KUKA KRL program: MyProgram_275().src

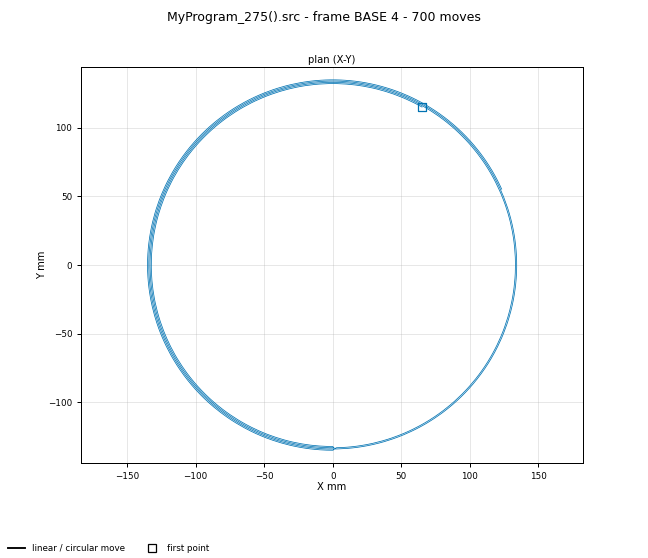
[picture p0: tool path of MyProgram_275().src in frame BASE 4, 700 of 700 moves have a stored position in this frame; points joined in program order, loops and branches not executed]
&ACCESS RVP
&REL 1
&PARAM TEMPLATE = C:\KRC\Roboter\Template\vorgabe
&PARAM EDITMASK = *
DEF MyProgram_275()
; ---- Setting reference (Base) ----
$BASE = BASE_DATA[4]

; --------------------------
; ---- Setting tool (TCP) ----
$TOOL = TOOL_DATA[3]
; --------------------------

$VEL.CP = VEL_APROX_PRINT
Startdeposition()
$VEL.CP = VEL_PRINT
LIN {X 65.127,Y 115.2291,Z 172,A 61.2414,B 9.2766,C 0.0638,E1 9.3556,E2 389.9841} C_DIS
LIN {X 62.4024,Y 116.727,Z 172,A 62.7582,B 9.2766,C 0.0584,E1 9.3518,E2 388.4469} C_DIS
LIN {X 59.3854,Y 118.2901,Z 172,A 64.0726,B 9.2766,C 0.0598,E1 9.3486,E2 387.151} C_DIS
LIN {X 56.4655,Y 119.7109,Z 172,A 65.4603,B 9.2766,C 0.0584,E1 9.3451,E2 385.7655} C_DIS
LIN {X 53.635,Y 121.0046,Z 172,A 66.8024,B 9.2766,C 0.0569,E1 9.3417,E2 384.424} C_DIS
LIN {X 50.5321,Y 122.3332,Z 172,A 68.2548,B 9.2766,C 0.0555,E1 9.3379,E2 382.9727} C_DIS
LIN {X 47.5119,Y 123.5374,Z 172,A 69.6526,B 9.2766,C 0.0543,E1 9.3343,E2 381.5762} C_DIS
LIN {X 44.4709,Y 124.6644,Z 172,A 71.05,B 9.2766,C 0.053,E1 9.3306,E2 380.1797} C_DIS
LIN {X 40.7766,Y 125.9215,Z 172,A 72.6186,B 9.2766,C 0.054,E1 9.3265,E2 378.6256} C_DIS
LIN {X 38.4338,Y 126.6555,Z 172,A 73.8215,B 9.2766,C 0.0503,E1 9.3232,E2 377.4063} C_DIS
LIN {X 35.3289,Y 127.5565,Z 172,A 75.1773,B 9.2766,C 0.0501,E1 9.3196,E2 376.056} C_DIS
LIN {X 32.2031,Y 128.3814,Z 172,A 76.5869,B 9.2767,C 0.0489,E1 9.3158,E2 374.6454} C_DIS
LIN {X 28.8757,Y 129.1715,Z 172,A 78.0434,B 9.2767,C 0.0484,E1 9.3118,E2 373.1922} C_DIS
LIN {X 25.6888,Y 129.8434,Z 172,A 79.4431,B 9.2767,C 0.0479,E1 9.308,E2 371.794} C_DIS
LIN {X 22.4953,Y 130.4347,Z 172,A 80.8231,B 9.2767,C 0.0477,E1 9.3042,E2 370.4175} C_DIS
LIN {X 19.425,Y 130.9271,Z 172,A 82.2366,B 9.2767,C 0.0458,E1 9.3003,E2 368.9965} C_DIS
LIN {X 16.2022,Y 131.364,Z 172,A 83.6161,B 9.2767,C 0.0458,E1 9.2965,E2 367.6208} C_DIS
LIN {X 12.5116,Y 131.7658,Z 172,A 85.1484,B 9.2767,C 0.0469,E1 9.2923,E2 366.0978} C_DIS
LIN {X 9.7365,Y 131.9999,Z 172,A 86.4152,B 9.2767,C 0.0455,E1 9.2887,E2 364.8243} C_DIS
LIN {X 6.4978,Y 132.199,Z 172,A 87.8269,B 9.2767,C 0.0451,E1 9.2848,E2 363.4123} C_DIS
LIN {X 3.2539,Y 132.3192,Z 172,A 89.2132,B 9.2767,C 0.0454,E1 9.2809,E2 362.0288} C_DIS
LIN {X 0.0153,Y 132.3605,Z 172,A 90.6902,B 9.2767,C 0.044,E1 9.2768,E2 360.5436} C_DIS
LIN {X -3.2492,Y 132.3193,Z 172,A 92.083,B 9.2767,C 0.0445,E1 9.2729,E2 359.1539} C_DIS
LIN {X -6.6259,Y 132.1926,Z 172,A 93.5018,B 9.2767,C 0.0456,E1 9.269,E2 357.7409} C_DIS
LIN {X -9.7303,Y 132.0004,Z 172,A 94.8665,B 9.2767,C 0.0456,E1 9.2651,E2 356.3748} C_DIS
LIN {X -13.1026,Y 131.7091,Z 172,A 96.308,B 9.2767,C 0.0464,E1 9.2612,E2 354.937} C_DIS
LIN {X -16.3389,Y 131.3477,Z 172,A 97.7167,B 9.2767,C 0.0469,E1 9.2572,E2 353.5291} C_DIS
LIN {X -19.5515,Y 130.9082,Z 172,A 99.1007,B 9.2767,C 0.0479,E1 9.2534,E2 352.1483} C_DIS
LIN {X -22.7528,Y 130.3893,Z 172,A 100.511,B 9.2767,C 0.0485,E1 9.2495,E2 350.7381} C_DIS
LIN {X -26.0765,Y 129.7645,Z 172,A 101.9358,B 9.2767,C 0.0501,E1 9.2457,E2 349.3187} C_DIS
LIN {X -29.4885,Y 129.0315,Z 172,A 103.4456,B 9.2767,C 0.0511,E1 9.2415,E2 347.81} C_DIS
LIN {X -32.29,Y 128.3594,Z 172,A 104.7854,B 9.2767,C 0.0503,E1 9.2379,E2 346.4602} C_DIS
LIN {X -35.9173,Y 127.392,Z 172,A 106.3281,B 9.2767,C 0.0531,E1 9.2338,E2 344.9283} C_DIS
LIN {X -38.4302,Y 126.6566,Z 172,A 107.5882,B 9.2767,C 0.0517,E1 9.2303,E2 343.654} C_DIS
LIN {X -41.6366,Y 125.6388,Z 172,A 108.9857,B 9.2767,C 0.0541,E1 9.2266,E2 342.2646} C_DIS
LIN {X -44.5824,Y 124.6241,Z 172,A 110.3733,B 9.2767,C 0.0548,E1 9.223,E2 340.8734} C_DIS
LIN {X -47.6183,Y 123.4961,Z 172,A 111.7823,B 9.2767,C 0.0561,E1 9.2193,E2 339.4646} C_DIS
LIN {X -50.7473,Y 122.2434,Z 172,A 113.2597,B 9.2767,C 0.0574,E1 9.2155,E2 337.9861} C_DIS
LIN {X -53.7595,Y 120.9489,Z 172,A 114.6384,B 9.2767,C 0.0598,E1 9.212,E2 336.6133} C_DIS
LIN {X -56.5897,Y 119.6516,Z 172,A 116.0384,B 9.2767,C 0.0606,E1 9.2084,E2 335.2083} C_DIS
LIN {X -59.5181,Y 118.2226,Z 172,A 117.496,B 9.2767,C 0.0616,E1 9.2048,E2 333.7464} C_DIS
LIN {X -62.5135,Y 116.6673,Z 172,A 118.9788,B 9.2767,C 0.0633,E1 9.2011,E2 332.2623} C_DIS
LIN {X -65.2363,Y 115.1675,Z 172,A 120.2908,B 9.2766,C 0.0658,E1 9.1979,E2 330.9554} C_DIS
LIN {X -68.1488,Y 113.4684,Z 172,A 121.7627,B 9.2766,C 0.0678,E1 9.1944,E2 329.4833} C_DIS
LIN {X -70.9084,Y 111.7643,Z 172,A 123.1624,B 9.2766,C 0.0701,E1 9.1911,E2 328.0853} C_DIS
LIN {X -74.0157,Y 109.731,Z 172,A 124.7159,B 9.2766,C 0.0736,E1 9.1875,E2 326.5396} C_DIS
LIN {X -76.2793,Y 108.1694,Z 172,A 125.9901,B 9.2766,C 0.0742,E1 9.1845,E2 325.2566} C_DIS
LIN {X -78.717,Y 106.4094,Z 172,A 127.4521,B 9.2766,C 0.0737,E1 9.1812,E2 323.7769} C_DIS
LIN {X -82.0673,Y 103.8473,Z 172,A 129.3252,B 9.2766,C 0.0762,E1 9.1771,E2 321.9} C_DIS
LIN {X -85.2696,Y 101.234,Z 172,A 131.1208,B 9.2765,C 0.0795,E1 9.1732,E2 320.1053} C_DIS
LIN {X -88.3376,Y 98.5679,Z 172,A 132.89,B 9.2765,C 0.0828,E1 9.1695,E2 318.3366} C_DIS
LIN {X -91.8024,Y 95.35,Z 172,A 134.8455,B 9.2765,C 0.0885,E1 9.1656,E2 316.3939} C_DIS
LIN {X -94.7344,Y 92.4374,Z 172,A 136.7676,B 9.2764,C 0.0899,E1 9.1618,E2 314.4579} C_DIS
LIN {X -97.5284,Y 89.484,Z 172,A 138.5544,B 9.2764,C 0.0933,E1 9.1584,E2 312.6697} C_DIS
LIN {X -100.2218,Y 86.4567,Z 172,A 140.3227,B 9.2764,C 0.0969,E1 9.1551,E2 310.9015} C_DIS
LIN {X -102.8625,Y 83.2979,Z 172,A 142.1311,B 9.2763,C 0.1005,E1 9.1519,E2 309.0918} C_DIS
LIN {X -105.4209,Y 80.0359,Z 172,A 143.7918,B 9.2763,C 0.107,E1 9.1491,E2 307.4488} C_DIS
LIN {X -107.2971,Y 77.5019,Z 172,A 145.1917,B 9.2762,C 0.1096,E1 9.1468,E2 306.0461} C_DIS
LIN {X -109.1538,Y 74.864,Z 172,A 146.6295,B 9.2762,C 0.1123,E1 9.1445,E2 304.6049} C_DIS
LIN {X -110.9486,Y 72.1775,Z 172,A 148.1,B 9.2762,C 0.1145,E1 9.1422,E2 303.1273} C_DIS
LIN {X -112.6772,Y 69.4484,Z 172,A 149.4685,B 9.2761,C 0.1185,E1 9.1402,E2 301.7638} C_DIS
LIN {X -114.4012,Y 66.5704,Z 172,A 150.9053,B 9.2761,C 0.1224,E1 9.1382,E2 300.3303} C_DIS
LIN {X -115.9291,Y 63.8724,Z 172,A 152.2877,B 9.276,C 0.1252,E1 9.1363,E2 298.9445} C_DIS
LIN {X -117.5491,Y 60.8396,Z 172,A 153.7952,B 9.276,C 0.1288,E1 9.1343,E2 297.4364} C_DIS
LIN {X -119.004,Y 57.941,Z 172,A 155.2177,B 9.2759,C 0.1321,E1 9.1326,E2 296.0131} C_DIS
LIN {X -120.3328,Y 55.1259,Z 172,A 156.5823,B 9.2759,C 0.1354,E1 9.131,E2 294.6479} C_DIS
LIN {X -121.6532,Y 52.1471,Z 172,A 158.0257,B 9.2759,C 0.1387,E1 9.1294,E2 293.2021} C_DIS
LIN {X -122.9461,Y 49.0219,Z 172,A 159.5002,B 9.2757,C 0.1425,E1 9.1278,E2 291.7279} C_DIS
LIN {X -124.1154,Y 45.981,Z 172,A 160.93,B 9.2757,C 0.146,E1 9.1264,E2 290.2972} C_DIS
LIN {X -125.2045,Y 42.9266,Z 172,A 162.3419,B 9.2757,C 0.1498,E1 9.1251,E2 288.8858} C_DIS
LIN {X -126.34,Y 39.4647,Z 172,A 163.9378,B 9.2756,C 0.1539,E1 9.1237,E2 287.2894} C_DIS
LIN {X -127.1202,Y 36.868,Z 172,A 165.147,B 9.2756,C 0.1566,E1 9.1228,E2 286.0771} C_DIS
LIN {X -127.9856,Y 33.7419,Z 172,A 166.5722,B 9.2755,C 0.1602,E1 9.1217,E2 284.6509} C_DIS
LIN {X -128.8049,Y 30.4681,Z 172,A 168.0566,B 9.2754,C 0.164,E1 9.1208,E2 283.1651} C_DIS
LIN {X -129.5239,Y 27.2532,Z 172,A 169.5788,B 9.2754,C 0.1665,E1 9.1199,E2 281.633} C_DIS
LIN {X -130.1092,Y 24.303,Z 172,A 170.8243,B 9.2753,C 0.1711,E1 9.1192,E2 280.3955} C_DIS
LIN {X -130.6809,Y 21.0199,Z 172,A 172.3104,B 9.2753,C 0.1746,E1 9.1185,E2 278.9057} C_DIS
LIN {X -131.1563,Y 17.8087,Z 172,A 173.7369,B 9.2751,C 0.1783,E1 9.118,E2 277.478} C_DIS
LIN {X -131.5527,Y 14.5881,Z 172,A 175.163,B 9.2751,C 0.182,E1 9.1175,E2 276.0508} C_DIS
LIN {X -131.8826,Y 11.214,Z 172,A 176.6177,B 9.275,C 0.1865,E1 9.1171,E2 274.599} C_DIS
LIN {X -132.1096,Y 8.1125,Z 172,A 178.0102,B 9.275,C 0.1896,E1 9.1169,E2 273.2023} C_DIS
LIN {X -132.2745,Y 4.7345,Z 172,A 179.4735,B 9.2748,C 0.1939,E1 9.1167,E2 271.7405} C_DIS
LIN {X -132.3534,Y 1.3457,Z 172,A -179.134,B 9.2748,C 0.1994,E1 9.1167,E2 270.3584} C_DIS
LIN {X -132.3475,Y -1.7648,Z 172,A -177.662,B 9.2747,C 0.2013,E1 9.1167,E2 268.8726} C_DIS
LIN {X -132.2638,Y -5.0086,Z 172,A -176.2074,B 9.2746,C 0.2045,E1 9.1167,E2 267.4133} C_DIS
LIN {X -132.0874,Y -8.4737,Z 172,A -174.7375,B 9.2745,C 0.2094,E1 9.117,E2 265.9486} C_DIS
LIN {X -131.8595,Y -11.4869,Z 172,A -173.3647,B 9.2745,C 0.2121,E1 9.1173,E2 264.5693} C_DIS
LIN {X -131.4649,Y -15.3568,Z 172,A -171.8356,B 9.2743,C 0.2195,E1 9.1178,E2 263.0602} C_DIS
LIN {X -131.1377,Y -17.9505,Z 172,A -170.4833,B 9.2743,C 0.2192,E1 9.1183,E2 261.6826} C_DIS
LIN {X -130.679,Y -21.0311,Z 172,A -169.0538,B 9.2743,C 0.2217,E1 9.1189,E2 260.2445} C_DIS
LIN {X -130.1175,Y -24.2591,Z 172,A -167.6784,B 9.2741,C 0.2264,E1 9.1196,E2 258.8755} C_DIS
LIN {X -129.4878,Y -27.4207,Z 172,A -166.2107,B 9.2741,C 0.2292,E1 9.1204,E2 257.4002} C_DIS
LIN {X -128.7496,Y -30.6976,Z 172,A -164.7876,B 9.2739,C 0.2338,E1 9.1213,E2 255.982} C_DIS
LIN {X -127.9636,Y -33.8244,Z 172,A -163.372,B 9.2739,C 0.2373,E1 9.1223,E2 254.5651} C_DIS
LIN {X -127.1019,Y -36.9304,Z 172,A -161.8377,B 9.2738,C 0.2389,E1 9.1235,E2 253.0151} C_DIS
LIN {X -125.7599,Y -41.2728,Z 172,A -159.8805,B 9.2736,C 0.2445,E1 9.1252,E2 251.0607} C_DIS
LIN {X -124.439,Y -45.0958,Z 172,A -158.2958,B 9.2734,C 0.252,E1 9.1266,E2 249.4973} C_DIS
LIN {X -123.3976,Y -47.8715,Z 172,A -156.8678,B 9.2734,C 0.253,E1 9.128,E2 248.0528} C_DIS
LIN {X -122.2317,Y -50.7753,Z 172,A -155.5005,B 9.2734,C 0.2564,E1 9.1295,E2 246.6849} C_DIS
LIN {X -120.9497,Y -53.7578,Z 172,A -154.0011,B 9.2733,C 0.2585,E1 9.1312,E2 245.1751} C_DIS
LIN {X -119.6466,Y -56.6002,Z 172,A -152.7067,B 9.2731,C 0.263,E1 9.1327,E2 243.8888} C_DIS
LIN {X -118.2264,Y -59.5107,Z 172,A -151.243,B 9.2731,C 0.2656,E1 9.1345,E2 242.4185} C_DIS
LIN {X -116.6748,Y -62.4995,Z 172,A -149.8397,B 9.2729,C 0.2702,E1 9.1363,E2 241.0228} C_DIS
LIN {X -115.1644,Y -65.2418,Z 172,A -148.4248,B 9.2729,C 0.2726,E1 9.1383,E2 239.6015} C_DIS
LIN {X -113.4581,Y -68.1657,Z 172,A -146.9417,B 9.2728,C 0.2759,E1 9.1404,E2 238.1171} C_DIS
LIN {X -111.7542,Y -70.9245,Z 172,A -145.3675,B 9.2728,C 0.2764,E1 9.1428,E2 236.523} C_DIS
LIN {X -109.9736,Y -73.6546,Z 172,A -144.085,B 9.2726,C 0.2819,E1 9.1447,E2 235.2568} C_DIS
LIN {X -107.9412,Y -76.6029,Z 172,A -142.5621,B 9.2725,C 0.2859,E1 9.1471,E2 233.738} C_DIS
LIN {X -106.316,Y -78.8425,Z 172,A -141.167,B 9.2725,C 0.2853,E1 9.1495,E2 232.3195} C_DIS
LIN {X -103.8545,Y -82.0582,Z 172,A -139.3643,B 9.2724,C 0.2884,E1 9.1526,E2 230.5116} C_DIS
LIN {X -101.2348,Y -85.2687,Z 172,A -137.5611,B 9.2723,C 0.2921,E1 9.1558,E2 228.708} C_DIS
LIN {X -98.5714,Y -88.3337,Z 172,A -135.9358,B 9.2721,C 0.2981,E1 9.1588,E2 227.0996} C_DIS
LIN {X -95.8719,Y -91.2568,Z 172,A -134.0515,B 9.2721,C 0.2988,E1 9.1624,E2 225.1962} C_DIS
LIN {X -92.9642,Y -94.2177,Z 172,A -132.2243,B 9.272,C 0.3018,E1 9.166,E2 223.3658} C_DIS
LIN {X -90.0913,Y -96.9677,Z 172,A -130.4908,B 9.2719,C 0.3049,E1 9.1696,E2 221.6314} C_DIS
LIN {X -87.0184,Y -99.7345,Z 172,A -128.7007,B 9.2718,C 0.3082,E1 9.1733,E2 219.8418} C_DIS
LIN {X -83.9207,Y -102.3549,Z 172,A -126.9148,B 9.2717,C 0.3108,E1 9.1772,E2 218.0527} C_DIS
LIN {X -80.3433,Y -105.1862,Z 172,A -125.0181,B 9.2715,C 0.3155,E1 9.1813,E2 216.166} C_DIS
LIN {X -77.5467,Y -107.2646,Z 172,A -123.5366,B 9.2715,C 0.3184,E1 9.1847,E2 214.6881} C_DIS
LIN {X -74.901,Y -109.1284,Z 172,A -122.1001,B 9.2714,C 0.32,E1 9.188,E2 213.2474} C_DIS
LIN {X -71.9097,Y -111.1224,Z 172,A -120.6166,B 9.2712,C 0.3236,E1 9.1914,E2 211.773} C_DIS
LIN {X -69.4334,Y -112.6864,Z 172,A -119.2487,B 9.2712,C 0.3236,E1 9.1947,E2 210.393} C_DIS
LIN {X -66.5381,Y -114.4199,Z 172,A -117.8103,B 9.2712,C 0.3261,E1 9.1981,E2 208.9574} C_DIS
LIN {X -63.0793,Y -116.3627,Z 172,A -115.9086,B 9.2712,C 0.3249,E1 9.2028,E2 207.0333} C_DIS
LIN {X -59.1058,Y -118.4294,Z 172,A -114.2002,B 9.271,C 0.3315,E1 9.207,E2 205.3531} C_DIS
LIN {X -56.4686,Y -119.7095,Z 172,A -112.8473,B 9.271,C 0.3315,E1 9.2104,E2 203.9899} C_DIS
LIN {X -53.6395,Y -121.0027,Z 172,A -111.4883,B 9.271,C 0.3326,E1 9.2139,E2 202.6293} C_DIS
LIN {X -50.5291,Y -122.3345,Z 172,A -110.0165,B 9.2709,C 0.334,E1 9.2177,E2 201.1565} C_DIS
LIN {X -47.5164,Y -123.5357,Z 172,A -108.603,B 9.2709,C 0.3351,E1 9.2214,E2 199.7417} C_DIS
LIN {X -43.7679,Y -124.9129,Z 172,A -107.016,B 9.2707,C 0.3393,E1 9.2255,E2 198.1718} C_DIS
LIN {X -41.5296,Y -125.6744,Z 172,A -105.8276,B 9.2707,C 0.337,E1 9.2287,E2 196.9631} C_DIS
LIN {X -38.447,Y -126.6515,Z 172,A -104.4389,B 9.2707,C 0.3383,E1 9.2324,E2 195.5755} C_DIS
LIN {X -35.3408,Y -127.5532,Z 172,A -103.029,B 9.2707,C 0.339,E1 9.2362,E2 194.1642} C_DIS
LIN {X -32.1624,Y -128.3918,Z 172,A -101.5669,B 9.2707,C 0.3392,E1 9.2402,E2 192.6969} C_DIS
LIN {X -28.8672,Y -129.1734,Z 172,A -100.1405,B 9.2707,C 0.3407,E1 9.244,E2 191.2751} C_DIS
LIN {X -25.6893,Y -129.8433,Z 172,A -98.736,B 9.2707,C 0.3414,E1 9.2479,E2 189.8703} C_DIS
LIN {X -22.5021,Y -130.4336,Z 172,A -97.3492,B 9.2706,C 0.3422,E1 9.2517,E2 188.4852} C_DIS
LIN {X -19.4209,Y -130.9277,Z 172,A -95.9517,B 9.2706,C 0.3418,E1 9.2556,E2 187.0814} C_DIS
LIN {X -16.1963,Y -131.3647,Z 172,A -94.5436,B 9.2706,C 0.3421,E1 9.2595,E2 185.6729} C_DIS
LIN {X -12.9725,Y -131.7216,Z 172,A -93.1122,B 9.2706,C 0.3418,E1 9.2635,E2 184.2377} C_DIS
LIN {X -9.7403,Y -131.9996,Z 172,A -91.7423,B 9.2706,C 0.3427,E1 9.2673,E2 182.8714} C_DIS
LIN {X -6.5025,Y -132.1988,Z 172,A -90.3296,B 9.2706,C 0.3426,E1 9.2712,E2 181.4571} C_DIS
LIN {X -3.2603,Y -132.319,Z 172,A -88.9419,B 9.2706,C 0.3428,E1 9.2751,E2 180.0709} C_DIS
LIN {X 0.0022,Y -132.3606,Z 172,A -87.4599,B 9.2706,C 0.3413,E1 9.2792,E2 178.5796} C_DIS
LIN {X 0.0022,Y -132.3606,Z 172,A -87.4599,B 9.2706,C 0.3413,E1 9.2792,E2 178.5796} C_DIS
Enddeposition()
LIN {X 0.9646,Y -133.2632,Z 172,A -87.4493,B 9.2704,C 0.3548,E1 9.2793,E2 178.6525} C_DIS
Startdeposition()
$VEL.CP = VEL_PRINT
LIN {X -2.4756,Y -133.245,Z 172,A -89.1713,B 9.2702,C 0.3597,E1 9.2744,E2 180.4051} C_DIS
LIN {X -6.4739,Y -133.1105,Z 172,A -90.8363,B 9.2702,C 0.3587,E1 9.2698,E2 182.0641} C_DIS
LIN {X -9.0906,Y -132.9586,Z 172,A -91.9518,B 9.2702,C 0.3584,E1 9.2667,E2 183.1787} C_DIS
LIN {X -11.5379,Y -132.7676,Z 172,A -93.049,B 9.2702,C 0.3591,E1 9.2636,E2 184.2814} C_DIS
LIN {X -14.6359,Y -132.462,Z 172,A -94.5024,B 9.2702,C 0.3611,E1 9.2595,E2 185.7494} C_DIS
LIN {X -18.1761,Y -132.0239,Z 172,A -95.9099,B 9.2702,C 0.3582,E1 9.2557,E2 187.142} C_DIS
LIN {X -21.515,Y -131.52,Z 172,A -97.4529,B 9.2702,C 0.3595,E1 9.2514,E2 188.6966} C_DIS
LIN {X -25.559,Y -130.7947,Z 172,A -99.3204,B 9.2702,C 0.3607,E1 9.2462,E2 190.577} C_DIS
LIN {X -29.5392,Y -129.9525,Z 172,A -100.9567,B 9.2702,C 0.3577,E1 9.2418,E2 192.2} C_DIS
LIN {X -33.0336,Y -129.1086,Z 172,A -102.5702,B 9.2702,C 0.3581,E1 9.2374,E2 193.8222} C_DIS
LIN {X -39.108,Y -127.4,Z 172,A -105.3268,B 9.2702,C 0.357,E1 9.23,E2 196.5845} C_DIS
LIN {X -42.5916,Y -126.279,Z 172,A -106.9251,B 9.2703,C 0.3563,E1 9.2257,E2 198.1862} C_DIS
LIN {X -47.3324,Y -124.5801,Z 172,A -108.9509,B 9.2705,C 0.3517,E1 9.2205,E2 200.1953} C_DIS
LIN {X -49.7048,Y -123.6511,Z 172,A -109.9688,B 9.2705,C 0.3492,E1 9.2179,E2 201.2037} C_DIS
LIN {X -52.1729,Y -122.6325,Z 172,A -111.2112,B 9.2705,C 0.3498,E1 9.2146,E2 202.4578} C_DIS
LIN {X -56.5524,Y -120.6749,Z 172,A -113.3293,B 9.2706,C 0.3486,E1 9.2092,E2 204.5828} C_DIS
LIN {X -61.9383,Y -117.999,Z 172,A -115.716,B 9.2709,C 0.3419,E1 9.2033,E2 206.9452} C_DIS
LIN {X -64.4835,Y -116.63,Z 172,A -117.2749,B 9.2707,C 0.346,E1 9.1994,E2 208.5427} C_DIS
LIN {X -68.5645,Y -114.2792,Z 172,A -119.1647,B 9.2709,C 0.3408,E1 9.1949,E2 210.4159} C_DIS
LIN {X -71.6191,Y -112.3897,Z 172,A -120.8881,B 9.2709,C 0.3418,E1 9.1908,E2 212.1609} C_DIS
LIN {X -76.7142,Y -108.9753,Z 172,A -123.3896,B 9.2711,C 0.3354,E1 9.185,E2 214.6456} C_DIS
LIN {X -79.3976,Y -107.0361,Z 172,A -124.8801,B 9.2711,C 0.3342,E1 9.1816,E2 216.1441} C_DIS
LIN {X -82.3345,Y -104.7935,Z 172,A -126.6316,B 9.2711,C 0.3344,E1 9.1777,E2 217.9149} C_DIS
LIN {X -85.5105,Y -102.2187,Z 172,A -128.3421,B 9.2713,C 0.3305,E1 9.1741,E2 219.6193} C_DIS
LIN {X -88.9556,Y -99.2349,Z 172,A -130.4345,B 9.2713,C 0.3292,E1 9.1697,E2 221.7272} C_DIS
LIN {X -92.6694,Y -95.776,Z 172,A -132.5765,B 9.2715,C 0.3243,E1 9.1653,E2 223.8637} C_DIS
LIN {X -95.8568,Y -92.586,Z 172,A -134.5288,B 9.2716,C 0.3207,E1 9.1615,E2 225.817} C_DIS
LIN {X -98.0931,Y -90.2131,Z 172,A -135.8736,B 9.2717,C 0.3168,E1 9.159,E2 227.1544} C_DIS
LIN {X -100.9844,Y -86.9644,Z 172,A -137.6298,B 9.2719,C 0.3109,E1 9.1558,E2 228.8961} C_DIS
LIN {X -103.337,Y -84.1556,Z 172,A -139.4124,B 9.2719,C 0.311,E1 9.1525,E2 230.7031} C_DIS
LIN {X -106.1013,Y -80.6432,Z 172,A -141.3567,B 9.2721,C 0.3071,E1 9.1492,E2 232.6493} C_DIS
LIN {X -108.7365,Y -77.0527,Z 172,A -143.2884,B 9.2721,C 0.303,E1 9.1461,E2 234.582} C_DIS
LIN {X -110.7148,Y -74.1818,Z 172,A -144.8304,B 9.2723,C 0.3002,E1 9.1436,E2 236.1284} C_DIS
LIN {X -113.1529,Y -70.4066,Z 172,A -146.6592,B 9.2725,C 0.2939,E1 9.1409,E2 237.9437} C_DIS
LIN {X -115.146,Y -67.0984,Z 172,A -148.3258,B 9.2726,C 0.2899,E1 9.1385,E2 239.6101} C_DIS
LIN {X -117.4363,Y -63.0031,Z 172,A -150.4071,B 9.2727,C 0.2859,E1 9.1357,E2 241.6978} C_DIS
LIN {X -119.008,Y -59.9792,Z 172,A -152.004,B 9.2727,C 0.2844,E1 9.1337,E2 243.3097} C_DIS
LIN {X -121.2219,Y -55.3693,Z 172,A -154.0796,B 9.273,C 0.2767,E1 9.1312,E2 245.369} C_DIS
LIN {X -122.4079,Y -52.6925,Z 172,A -155.3909,B 9.273,C 0.2742,E1 9.1298,E2 246.6857} C_DIS
LIN {X -124.0169,Y -48.7879,Z 172,A -157.2911,B 9.2732,C 0.2708,E1 9.1278,E2 248.5948} C_DIS
LIN {X -125.6242,Y -44.4892,Z 172,A -159.2098,B 9.2734,C 0.2646,E1 9.1259,E2 250.5056} C_DIS
LIN {X -126.5759,Y -41.7,Z 172,A -160.523,B 9.2734,C 0.2619,E1 9.1248,E2 251.8233} C_DIS
LIN {X -127.931,Y -37.3342,Z 172,A -162.8222,B 9.2734,C 0.2619,E1 9.1229,E2 254.1609} C_DIS
LIN {X -128.8278,Y -34.1119,Z 172,A -164.5855,B 9.2734,C 0.2631,E1 9.1216,E2 255.9617} C_DIS
LIN {X -129.9932,Y -29.361,Z 172,A -165.9012,B 9.2739,C 0.2445,E1 9.1208,E2 257.1819} C_DIS
LIN {X -131.253,Y -23.0871,Z 172,A -168.8496,B 9.274,C 0.2399,E1 9.1192,E2 260.1517} C_DIS
LIN {X -131.7541,Y -20.0301,Z 172,A -170.1937,B 9.2741,C 0.2363,E1 9.1186,E2 261.4961} C_DIS
LIN {X -132.2024,Y -16.823,Z 172,A -171.7869,B 9.2741,C 0.2356,E1 9.118,E2 263.1121} C_DIS
LIN {X -132.7024,Y -12.2694,Z 172,A -173.7422,B 9.2743,C 0.2297,E1 9.1175,E2 265.064} C_DIS
LIN {X -133.0031,Y -8.396,Z 172,A -175.3974,B 9.2744,C 0.2246,E1 9.1172,E2 266.7159} C_DIS
LIN {X -133.1956,Y -4.4468,Z 172,A -177.0496,B 9.2745,C 0.2189,E1 9.117,E2 268.3608} C_DIS
LIN {X -133.2611,Y -1.5053,Z 172,A -178.4647,B 9.2745,C 0.2176,E1 9.117,E2 269.7927} C_DIS
LIN {X -133.2378,Y 2.9053,Z 172,A 179.7323,B 9.2747,C 0.2106,E1 9.117,E2 271.5828} C_DIS
LIN {X -133.1018,Y 6.6476,Z 172,A 178.021,B 9.2748,C 0.2076,E1 9.1172,E2 273.3045} C_DIS
LIN {X -132.8607,Y 10.4323,Z 172,A 176.2293,B 9.2748,C 0.2054,E1 9.1175,E2 275.1138} C_DIS
LIN {X -132.4694,Y 14.5669,Z 172,A 174.5942,B 9.275,C 0.1978,E1 9.118,E2 276.7292} C_DIS
LIN {X -132.1331,Y 17.3514,Z 172,A 173.343,B 9.275,C 0.1951,E1 9.1184,E2 277.9846} C_DIS
LIN {X -131.5777,Y 21.169,Z 172,A 171.1413,B 9.275,C 0.199,E1 9.1194,E2 280.2489} C_DIS
LIN {X -130.8179,Y 25.4374,Z 172,A 169.8293,B 9.2753,C 0.1848,E1 9.1201,E2 281.4938} C_DIS
LIN {X -130.1385,Y 28.7147,Z 172,A 168.1357,B 9.2753,C 0.1848,E1 9.1211,E2 283.2162} C_DIS
LIN {X -129.1205,Y 32.9867,Z 172,A 166.302,B 9.2754,C 0.1786,E1 9.1223,E2 285.0414} C_DIS
LIN {X -128.1784,Y 36.481,Z 172,A 164.8579,B 9.2755,C 0.1724,E1 9.1234,E2 286.4707} C_DIS
LIN {X -127.2073,Y 39.7375,Z 172,A 163.3411,B 9.2755,C 0.1692,E1 9.1246,E2 287.9926} C_DIS
LIN {X -126.3231,Y 42.459,Z 172,A 162.1334,B 9.2756,C 0.1654,E1 9.1257,E2 289.1963} C_DIS
LIN {X -125.0854,Y 45.9831,Z 172,A 160.2736,B 9.2756,C 0.1651,E1 9.1274,E2 291.0845} C_DIS
LIN {X -123.9028,Y 49.0803,Z 172,A 158.8706,B 9.2757,C 0.1609,E1 9.1289,E2 292.4835} C_DIS
LIN {X -122.2751,Y 52.9995,Z 172,A 157.1666,B 9.2758,C 0.154,E1 9.1307,E2 294.1712} C_DIS
LIN {X -120.6012,Y 56.7111,Z 172,A 155.3929,B 9.2759,C 0.1497,E1 9.1328,E2 295.946} C_DIS
LIN {X -119.3293,Y 59.3366,Z 172,A 154.0415,B 9.2759,C 0.148,E1 9.1345,E2 297.3074} C_DIS
LIN {X -117.6722,Y 62.5607,Z 172,A 152.2216,B 9.2759,C 0.1482,E1 9.1369,E2 299.1565} C_DIS
LIN {X -116.0917,Y 65.4478,Z 172,A 150.9338,B 9.276,C 0.1425,E1 9.1386,E2 300.4278} C_DIS
LIN {X -113.4285,Y 69.9625,Z 172,A 148.9639,B 9.2762,C 0.1322,E1 9.1414,E2 302.3619} C_DIS
LIN {X -111.8526,Y 72.4546,Z 172,A 147.4781,B 9.2762,C 0.1327,E1 9.1436,E2 303.8722} C_DIS
LIN {X -107.9778,Y 78.1119,Z 172,A 144.5538,B 9.2762,C 0.1252,E1 9.1483,E2 306.7906} C_DIS
LIN {X -105.6332,Y 81.2552,Z 172,A 142.6957,B 9.2762,C 0.1241,E1 9.1514,E2 308.6674} C_DIS
LIN {X -102.9074,Y 84.6811,Z 172,A 140.9071,B 9.2764,C 0.1182,E1 9.1546,E2 310.443} C_DIS
LIN {X -100.6071,Y 87.4011,Z 172,A 139.2363,B 9.2764,C 0.1171,E1 9.1576,E2 312.1287} C_DIS
LIN {X -97.4626,Y 90.8939,Z 172,A 137.2199,B 9.2764,C 0.1126,E1 9.1614,E2 314.1425} C_DIS
LIN {X -94.3493,Y 94.1219,Z 172,A 135.2794,B 9.2764,C 0.1088,E1 9.1652,E2 316.0826} C_DIS
LIN {X -91.5455,Y 96.8509,Z 172,A 133.6704,B 9.2765,C 0.1041,E1 9.1684,E2 317.6813} C_DIS
LIN {X -88.5666,Y 99.583,Z 172,A 131.8128,B 9.2765,C 0.1027,E1 9.1723,E2 319.5513} C_DIS
LIN {X -85.2789,Y 102.4124,Z 172,A 129.9379,B 9.2765,C 0.0993,E1 9.1763,E2 321.4256} C_DIS
LIN {X -82.1778,Y 104.9166,Z 172,A 127.0716,B 9.2764,C 0.1157,E1 9.183,E2 324.4241} C_DIS
LIN {X -75.7351,Y 109.6586,Z 172,A 124.8388,B 9.2767,C 0.0894,E1 9.1877,E2 326.5138} C_DIS
LIN {X -72.5416,Y 111.7961,Z 172,A 123.1434,B 9.2767,C 0.0874,E1 9.1916,E2 328.2127} C_DIS
LIN {X -69.1847,Y 113.9044,Z 172,A 121.3147,B 9.2767,C 0.0869,E1 9.196,E2 330.0546} C_DIS
LIN {X -65.1267,Y 116.2722,Z 172,A 119.3051,B 9.2767,C 0.0837,E1 9.2009,E2 332.0612} C_DIS
LIN {X -61.054,Y 118.4609,Z 172,A 117.4661,B 9.2767,C 0.0784,E1 9.2054,E2 333.8811} C_DIS
LIN {X -57.7742,Y 120.0933,Z 172,A 115.9971,B 9.2768,C 0.0744,E1 9.209,E2 335.3362} C_DIS
LIN {X -55.188,Y 121.3058,Z 172,A 114.5797,B 9.2768,C 0.0763,E1 9.2127,E2 336.7751} C_DIS
LIN {X -51.887,Y 122.7526,Z 172,A 112.4244,B 9.2768,C 0.0852,E1 9.2184,E2 338.9998} C_DIS
LIN {X -47.4476,Y 124.5369,Z 172,A 110.981,B 9.2768,C 0.0721,E1 9.222,E2 340.3701} C_DIS
LIN {X -44.4503,Y 125.6382,Z 172,A 109.5817,B 9.2768,C 0.0711,E1 9.2256,E2 341.7714} C_DIS
LIN {X -40.0878,Y 127.0959,Z 172,A 107.6057,B 9.2768,C 0.0693,E1 9.2309,E2 343.7458} C_DIS
LIN {X -35.1727,Y 128.5442,Z 172,A 105.3797,B 9.2768,C 0.0679,E1 9.2368,E2 345.973} C_DIS
LIN {X -32.6355,Y 129.2096,Z 172,A 104.2212,B 9.2768,C 0.0676,E1 9.24,E2 347.1343} C_DIS
LIN {X -29.6558,Y 129.9259,Z 172,A 102.8913,B 9.2768,C 0.0669,E1 9.2436,E2 348.4647} C_DIS
LIN {X -25.9596,Y 130.7161,Z 172,A 101.1296,B 9.2768,C 0.0684,E1 9.2485,E2 350.2415} C_DIS
LIN {X -22.1207,Y 131.4189,Z 172,A 99.5355,B 9.2768,C 0.066,E1 9.2528,E2 351.8247} C_DIS
LIN {X -18.3687,Y 131.9964,Z 172,A 98.0008,B 9.2768,C 0.0634,E1 9.257,E2 353.3471} C_DIS
LIN {X -14.9248,Y 132.4309,Z 172,A 96.3394,B 9.2768,C 0.066,E1 9.2617,E2 355.0275} C_DIS
LIN {X -10.7054,Y 132.8379,Z 172,A 94.4825,B 9.2768,C 0.0662,E1 9.2669,E2 356.8874} C_DIS
LIN {X -6.5116,Y 133.1086,Z 172,A 92.7561,B 9.2768,C 0.0643,E1 9.2716,E2 358.6035} C_DIS
LIN {X -2.0749,Y 133.2516,Z 172,A 90.9085,B 9.2768,C 0.063,E1 9.2768,E2 360.443} C_DIS
LIN {X 2.1724,Y 133.25,Z 172,A 89.0609,B 9.2768,C 0.0634,E1 9.2819,E2 362.2923} C_DIS
LIN {X 5.6401,Y 133.149,Z 172,A 87.6427,B 9.2769,C 0.0621,E1 9.2859,E2 363.7013} C_DIS
LIN {X 8.9084,Y 132.9715,Z 172,A 86.0546,B 9.2769,C 0.0658,E1 9.2904,E2 365.3101} C_DIS
LIN {X 12.899,Y 132.642,Z 172,A 84.4461,B 9.2769,C 0.064,E1 9.2948,E2 366.9047} C_DIS
LIN {X 16.3625,Y 132.2605,Z 172,A 82.8167,B 9.2769,C 0.067,E1 9.2994,E2 368.549} C_DIS
LIN {X 21.1297,Y 131.5839,Z 172,A 80.9417,B 9.2769,C 0.0641,E1 9.3045,E2 370.4004} C_DIS
LIN {X 24.2201,Y 131.0503,Z 172,A 79.5943,B 9.2769,C 0.0647,E1 9.3082,E2 371.7474} C_DIS
LIN {X 26.5698,Y 130.5919,Z 172,A 78.5498,B 9.2769,C 0.0655,E1 9.311,E2 372.7933} C_DIS
LIN {X 29.9187,Y 129.8658,Z 172,A 77.0367,B 9.2769,C 0.0672,E1 9.3152,E2 374.3108} C_DIS
LIN {X 35.966,Y 128.3224,Z 172,A 74.2415,B 9.2769,C 0.0714,E1 9.3228,E2 377.1186} C_DIS
LIN {X 39.6366,Y 127.2382,Z 172,A 72.6283,B 9.2769,C 0.0721,E1 9.3271,E2 378.7278} C_DIS
LIN {X 44.3497,Y 125.6734,Z 172,A 70.6589,B 9.2769,C 0.0707,E1 9.3322,E2 380.6775} C_DIS
LIN {X 46.7108,Y 124.8129,Z 172,A 69.538,B 9.2769,C 0.0726,E1 9.3352,E2 381.8029} C_DIS
LIN {X 49.9361,Y 123.5579,Z 172,A 68.0967,B 9.2769,C 0.0732,E1 9.3389,E2 383.2386} C_DIS
LIN {X 53.6578,Y 121.9904,Z 172,A 66.3671,B 9.2769,C 0.075,E1 9.3433,E2 384.9675} C_DIS
LIN {X 57.6789,Y 120.1388,Z 172,A 64.4536,B 9.2768,C 0.0775,E1 9.3482,E2 386.882} C_DIS
LIN {X 60.8786,Y 118.5502,Z 172,A 62.886,B 9.2768,C 0.0801,E1 9.3521,E2 388.4534} C_DIS
LIN {X 64.8754,Y 116.4129,Z 172,A 61.0878,B 9.2768,C 0.0797,E1 9.3565,E2 390.234} C_DIS
LIN {X 67.8909,Y 114.6806,Z 172,A 59.4057,B 9.2768,C 0.0857,E1 9.3606,E2 391.9383} C_DIS
LIN {X 71.817,Y 112.263,Z 172,A 56.5973,B 9.2765,C 0.1058,E1 9.3674,E2 394.8439} C_DIS
LIN {X 77.4097,Y 108.4823,Z 172,A 54.6563,B 9.2767,C 0.0906,E1 9.3716,E2 396.6725} C_DIS
LIN {X 81.3117,Y 105.5899,Z 172,A 52.7782,B 9.2767,C 0.0897,E1 9.3757,E2 398.526} C_DIS
LIN {X 83.5184,Y 103.8526,Z 172,A 51.3083,B 9.2766,C 0.0974,E1 9.379,E2 400.0274} C_DIS
LIN {X 87.0731,Y 100.8908,Z 172,A 49.1318,B 9.2766,C 0.1051,E1 9.3837,E2 402.2266} C_DIS
LIN {X 89.5926,Y 98.6601,Z 172,A 48.1248,B 9.2766,C 0.0985,E1 9.3857,E2 403.1818} C_DIS
LIN {X 92.1781,Y 96.249,Z 172,A 46.4262,B 9.2766,C 0.1053,E1 9.3892,E2 404.9022} C_DIS
LIN {X 96.5286,Y 91.8856,Z 172,A 44.029,B 9.2766,C 0.1053,E1 9.3938,E2 407.2702} C_DIS
LIN {X 98.8565,Y 89.3762,Z 172,A 42.3652,B 9.2764,C 0.1126,E1 9.397,E2 408.9576} C_DIS
LIN {X 101.453,Y 86.4173,Z 172,A 39.8737,B 9.2762,C 0.1334,E1 9.4017,E2 411.5442} C_DIS
LIN {X 105.4967,Y 81.4321,Z 172,A 38.224,B 9.2764,C 0.1157,E1 9.4043,E2 413.0637} C_DIS
LIN {X 109.2448,Y 76.3303,Z 172,A 35.4493,B 9.2763,C 0.1232,E1 9.4089,E2 415.8461} C_DIS
LIN {X 111.0216,Y 73.7222,Z 172,A 33.8944,B 9.2762,C 0.1308,E1 9.4113,E2 417.4254} C_DIS
LIN {X 113.2937,Y 70.1803,Z 172,A 32.1369,B 9.2762,C 0.1341,E1 9.414,E2 419.1778} C_DIS
LIN {X 115.1371,Y 67.1138,Z 172,A 30.5859,B 9.2761,C 0.1381,E1 9.4162,E2 420.7312} C_DIS
LIN {X 117.0478,Y 63.722,Z 172,A 28.9463,B 9.2761,C 0.1416,E1 9.4184,E2 422.3677} C_DIS
LIN {X 118.7634,Y 60.4598,Z 172,A 27.4063,B 9.276,C 0.1447,E1 9.4203,E2 423.9033} C_DIS
LIN {X 120.5874,Y 56.74,Z 172,A 25.7518,B 9.276,C 0.1465,E1 9.4223,E2 425.5438} C_DIS
LIN {X 121.7109,Y 54.2827,Z 172,A 24.5585,B 9.2759,C 0.1503,E1 9.4237,E2 426.7417} C_DIS
LIN {X 123.2343,Y 50.7337,Z 172,A 22.9991,B 9.2759,C 0.1524,E1 9.4254,E2 428.2901} C_DIS
LIN {X 125.1577,Y 45.783,Z 172,A 20.7986,B 9.2758,C 0.1568,E1 9.4276,E2 430.4823} C_DIS
LIN {X 126.2158,Y 42.7814,Z 172,A 19.2481,B 9.2757,C 0.1646,E1 9.429,E2 432.0558} C_DIS
LIN {X 127.8977,Y 37.448,Z 172,A 17.0598,B 9.2757,C 0.1664,E1 9.4308,E2 434.2198} C_DIS
LIN {X 128.7599,Y 34.3668,Z 172,A 15.6603,B 9.2755,C 0.1707,E1 9.4318,E2 435.6234} C_DIS
LIN {X 129.5766,Y 31.1465,Z 172,A 14.2354,B 9.2755,C 0.1747,E1 9.4328,E2 437.049} C_DIS
LIN {X 130.3959,Y 27.5225,Z 172,A 12.6777,B 9.2755,C 0.1783,E1 9.4337,E2 438.6033} C_DIS
LIN {X 130.9549,Y 24.721,Z 172,A 11.3685,B 9.2753,C 0.1836,E1 9.4344,E2 439.9232} C_DIS
LIN {X 131.7003,Y 20.3781,Z 172,A 9.5864,B 9.2753,C 0.1865,E1 9.4352,E2 441.6934} C_DIS
LIN {X 132.2081,Y 16.7791,Z 172,A 7.9113,B 9.2751,C 0.1935,E1 9.4358,E2 443.3835} C_DIS
LIN {X 132.6483,Y 12.8333,Z 172,A 6.2865,B 9.2751,C 0.1966,E1 9.4363,E2 444.9998} C_DIS
LIN {X 132.9754,Y 8.8443,Z 172,A 4.7502,B 9.2751,C 0.1974,E1 9.4366,E2 446.5155} C_DIS
LIN {X 133.1414,Y 5.836,Z 172,A 3.2408,B 9.2748,C 0.206,E1 9.4368,E2 448.052} C_DIS
LIN {X 133.2647,Y 1.0317,Z 172,A 1.3333,B 9.2748,C 0.2085,E1 9.4369,E2 449.9422} C_DIS
LIN {X 133.2347,Y -3.0379,Z 172,A -0.2858,B 9.2748,C 0.2106,E1 9.4369,E2 451.5472} C_DIS
LIN {X 133.1391,Y -5.8956,Z 172,A -1.7326,B 9.2745,C 0.2191,E1 9.4367,E2 453.0215} C_DIS
LIN {X 132.9195,Y -9.627,Z 172,A -3.156,B 9.2745,C 0.2196,E1 9.4364,E2 454.4242} C_DIS
LIN {X 132.61,Y -13.2316,Z 172,A -4.6176,B 9.2745,C 0.222,E1 9.4361,E2 455.876} C_DIS
LIN {X 132.275,Y -16.2413,Z 172,A -5.9141,B 9.2744,C 0.2257,E1 9.4356,E2 457.1731} C_DIS
LIN {X 131.9171,Y -18.9237,Z 172,A -7.0998,B 9.2743,C 0.2295,E1 9.4352,E2 458.3627} C_DIS
LIN {X 131.2903,Y -22.8791,Z 172,A -8.9076,B 9.2741,C 0.2364,E1 9.4343,E2 460.1826} C_DIS
LIN {X 130.5598,Y -26.7276,Z 172,A -10.4961,B 9.2741,C 0.2391,E1 9.4335,E2 461.7613} C_DIS
LIN {X 129.156,Y -32.847,Z 172,A -13.8223,B 9.2735,C 0.2609,E1 9.4312,E2 465.1659} C_DIS
LIN {X 127.6755,Y -38.2067,Z 172,A -15.454,B 9.2738,C 0.2506,E1 9.43,E2 466.7084} C_DIS
LIN {X 126.134,Y -43.0213,Z 172,A -17.541,B 9.2736,C 0.2547,E1 9.4283,E2 468.7872} C_DIS
LIN {X 125.2999,Y -45.3886,Z 172,A -18.6637,B 9.2736,C 0.2587,E1 9.4272,E2 469.9163} C_DIS
LIN {X 124.2037,Y -48.3073,Z 172,A -20.0871,B 9.2734,C 0.2642,E1 9.4257,E2 471.3513} C_DIS
LIN {X 122.4126,Y -52.6816,Z 172,A -22.794,B 9.2728,C 0.2848,E1 9.4227,E2 474.1419} C_DIS
LIN {X 119.9059,Y -58.1665,Z 172,A -24.5455,B 9.2731,C 0.273,E1 9.4207,E2 475.7944} C_DIS
LIN {X 118.589,Y -60.8023,Z 172,A -25.7996,B 9.2731,C 0.276,E1 9.4191,E2 477.0482} C_DIS
LIN {X 116.8024,Y -64.1719,Z 172,A -27.7456,B 9.2727,C 0.2872,E1 9.4165,E2 479.0333} C_DIS
LIN {X 115.1026,Y -67.1728,Z 172,A -28.916,B 9.2727,C 0.284,E1 9.4149,E2 480.1673} C_DIS
LIN {X 113.0039,Y -70.6459,Z 172,A -30.6046,B 9.2727,C 0.2872,E1 9.4124,E2 481.8509} C_DIS
LIN {X 110.8253,Y -74.0163,Z 172,A -32.491,B 9.2725,C 0.2951,E1 9.4095,E2 483.7587} C_DIS
LIN {X 108.771,Y -77.0038,Z 172,A -33.8438,B 9.2725,C 0.2943,E1 9.4074,E2 485.088} C_DIS
LIN {X 106.7724,Y -79.7519,Z 172,A -35.2874,B 9.2724,C 0.2974,E1 9.405,E2 486.5311} C_DIS
LIN {X 104.373,Y -82.8671,Z 172,A -37.0214,B 9.2722,C 0.3024,E1 9.402,E2 488.2721} C_DIS
LIN {X 99.8049,Y -88.3156,Z 172,A -39.8457,B 9.2722,C 0.3042,E1 9.397,E2 491.0711} C_DIS
LIN {X 97.5266,Y -90.8253,Z 172,A -41.4846,B 9.2719,C 0.3115,E1 9.3938,E2 492.7338} C_DIS
LIN {X 94.3812,Y -94.0899,Z 172,A -43.9364,B 9.2714,C 0.3266,E1 9.3889,E2 495.2487} C_DIS
LIN {X 90.8717,Y -97.4833,Z 172,A -45.2744,B 9.2718,C 0.3144,E1 9.3863,E2 496.496} C_DIS
LIN {X 88.9333,Y -99.2549,Z 172,A -46.6081,B 9.2716,C 0.3212,E1 9.3835,E2 497.856} C_DIS
LIN {X 85.6284,Y -102.1197,Z 172,A -48.4453,B 9.2715,C 0.324,E1 9.3796,E2 499.6897} C_DIS
LIN {X 80.9694,Y -105.8519,Z 172,A -50.9955,B 9.2713,C 0.3285,E1 9.374,E2 502.2404} C_DIS
LIN {X 77.5248,Y -108.4,Z 172,A -52.9144,B 9.2712,C 0.3334,E1 9.3697,E2 504.1704} C_DIS
LIN {X 74.4424,Y -110.54,Z 172,A -54.4113,B 9.2712,C 0.3337,E1 9.3663,E2 505.6547} C_DIS
LIN {X 70.78,Y -112.9204,Z 172,A -56.7374,B 9.2707,C 0.3464,E1 9.3606,E2 508.0372} C_DIS
LIN {X 66.9538,Y -115.2297,Z 172,A -58.6059,B 9.2707,C 0.3483,E1 9.3561,E2 509.901} C_DIS
LIN {X 63.201,Y -117.33,Z 172,A -59.9644,B 9.2709,C 0.3407,E1 9.3529,E2 511.2011} C_DIS
LIN {X 58.3131,Y -119.8342,Z 172,A -62.2701,B 9.2709,C 0.3429,E1 9.3472,E2 513.5021} C_DIS
LIN {X 55.7824,Y -121.0309,Z 172,A -63.575,B 9.2707,C 0.3466,E1 9.3439,E2 514.8203} C_DIS
LIN {X 52.1961,Y -122.6225,Z 172,A -65.3161,B 9.2706,C 0.3499,E1 9.3394,E2 516.5696} C_DIS
LIN {X 48.2504,Y -124.2258,Z 172,A -67.7359,B 9.27,C 0.3642,E1 9.3329,E2 519.0624} C_DIS
LIN {X 42.8408,Y -126.1952,Z 172,A -69.4559,B 9.2705,C 0.3513,E1 9.3286,E2 520.6924} C_DIS
LIN {X 40.2544,Y -127.0427,Z 172,A -70.6232,B 9.2705,C 0.3524,E1 9.3255,E2 521.8602} C_DIS
LIN {X 35.9901,Y -128.3156,Z 172,A -72.6052,B 9.2703,C 0.3556,E1 9.3202,E2 523.8519} C_DIS
LIN {X 31.9272,Y -129.3884,Z 172,A -74.2523,B 9.2704,C 0.3538,E1 9.3157,E2 525.4807} C_DIS
LIN {X 29.3679,Y -129.9916,Z 172,A -75.4482,B 9.2704,C 0.356,E1 9.3125,E2 526.6854} C_DIS
LIN {X 25.2521,Y -130.8533,Z 172,A -77.2449,B 9.2703,C 0.3571,E1 9.3075,E2 528.4819} C_DIS
LIN {X 21.2817,Y -131.5589,Z 172,A -78.9413,B 9.2703,C 0.3574,E1 9.3029,E2 530.1749} C_DIS
LIN {X 17.4875,Y -132.1153,Z 172,A -80.6049,B 9.2703,C 0.3585,E1 9.2983,E2 531.8412} C_DIS
LIN {X 13.8577,Y -132.5457,Z 172,A -82.1576,B 9.2703,C 0.3589,E1 9.294,E2 533.3926} C_DIS
LIN {X 10.5947,Y -132.8473,Z 172,A -83.723,B 9.2701,C 0.3625,E1 9.2896,E2 534.978} C_DIS
LIN {X 6.5867,Y -133.1048,Z 172,A -85.3476,B 9.2701,C 0.361,E1 9.2851,E2 536.5909} C_DIS
LIN {X 2.7736,Y -133.24,Z 172,A -86.8252,B 9.2703,C 0.3581,E1 9.281,E2 538.0495} C_DIS
LIN {X 2.7736,Y -133.24,Z 172,A -86.8252,B 9.2703,C 0.3581,E1 9.281,E2 538.0495} C_DIS
Enddeposition()
LIN {X 0.9679,Y -134.1726,Z 172,A -87.54,B 9.2701,C 0.3625,E1 9.2789,E2 538.7911} C_DIS
Startdeposition()
$VEL.CP = VEL_PRINT
LIN {X 3.458,Y -134.1325,Z 172,A -86.008,B 9.2705,C 0.3529,E1 9.2834,E2 537.2003} C_DIS
LIN {X 8.321,Y -133.9185,Z 172,A -83.8917,B 9.2705,C 0.3515,E1 9.2893,E2 535.0782} C_DIS
LIN {X 11.0041,Y -133.7251,Z 172,A -82.4409,B 9.2708,C 0.3449,E1 9.2934,E2 533.5889} C_DIS
LIN {X 14.3084,Y -133.4116,Z 172,A -81.3277,B 9.2705,C 0.3506,E1 9.2964,E2 532.513} C_DIS
LIN {X 18.2622,Y -132.93,Z 172,A -79.5804,B 9.2706,C 0.3488,E1 9.3013,E2 530.759} C_DIS
LIN {X 22.1248,Y -132.3399,Z 172,A -78.0103,B 9.2706,C 0.3499,E1 9.3056,E2 529.2001} C_DIS
LIN {X 25.5802,Y -131.7162,Z 172,A -76.3488,B 9.2707,C 0.3455,E1 9.3102,E2 527.5173} C_DIS
LIN {X 29.7346,Y -130.8404,Z 172,A -74.6033,B 9.2707,C 0.3455,E1 9.3149,E2 525.7791} C_DIS
LIN {X 34.1398,Y -129.7613,Z 172,A -72.6837,B 9.2707,C 0.3443,E1 9.3201,E2 523.8603} C_DIS
LIN {X 37.5202,Y -128.8239,Z 172,A -71.2247,B 9.2707,C 0.3437,E1 9.324,E2 522.4051} C_DIS
LIN {X 41.0236,Y -127.7514,Z 172,A -69.6791,B 9.2708,C 0.3426,E1 9.3282,E2 520.8607} C_DIS
LIN {X 43.6763,Y -126.8691,Z 172,A -68.1264,B 9.2712,C 0.3337,E1 9.3324,E2 519.262} C_DIS
LIN {X 47.2138,Y -125.5953,Z 172,A -66.8576,B 9.271,C 0.3391,E1 9.3356,E2 518.0343} C_DIS
LIN {X 51.4372,Y -123.9257,Z 172,A -65.1018,B 9.271,C 0.3407,E1 9.3401,E2 516.3} C_DIS
LIN {X 54.5674,Y -122.5795,Z 172,A -63.5215,B 9.271,C 0.3361,E1 9.3442,E2 514.7028} C_DIS
LIN {X 57.157,Y -121.3957,Z 172,A -62.3778,B 9.271,C 0.3361,E1 9.347,E2 513.5673} C_DIS
LIN {X 60.5419,Y -119.7418,Z 172,A -60.7731,B 9.2712,C 0.3339,E1 9.3511,E2 511.9616} C_DIS
LIN {X 64.0054,Y -117.9282,Z 172,A -58.6068,B 9.2716,C 0.3206,E1 9.3566,E2 509.7314} C_DIS
LIN {X 67.7551,Y -115.815,Z 172,A -56.9822,B 9.2716,C 0.3224,E1 9.3604,E2 508.1321} C_DIS
LIN {X 70.5468,Y -114.1364,Z 172,A -55.7868,B 9.2715,C 0.3244,E1 9.3632,E2 506.96} C_DIS
LIN {X 74.0687,Y -111.8828,Z 172,A -54.0307,B 9.2715,C 0.3221,E1 9.3673,E2 505.206} C_DIS
LIN {X 78.687,Y -108.6838,Z 172,A -51.8006,B 9.2715,C 0.3216,E1 9.3724,E2 502.9949} C_DIS
LIN {X 80.8914,Y -107.0533,Z 172,A -50.0563,B 9.2721,C 0.3067,E1 9.3764,E2 501.1774} C_DIS
LIN {X 84.4667,Y -104.2558,Z 172,A -48.5839,B 9.2719,C 0.3134,E1 9.3795,E2 499.7618} C_DIS
LIN {X 87.696,Y -101.5542,Z 172,A -46.7832,B 9.2719,C 0.3098,E1 9.3833,E2 497.9589} C_DIS
LIN {X 91.13,Y -98.485,Z 172,A -45.0762,B 9.2719,C 0.3115,E1 9.3868,E2 496.2826} C_DIS
LIN {X 93.7751,Y -95.9685,Z 172,A -43.318,B 9.2722,C 0.3038,E1 9.3904,E2 494.4978} C_DIS
LIN {X 96.7912,Y -92.9267,Z 172,A -41.4835,B 9.2723,C 0.2997,E1 9.3939,E2 492.6609} C_DIS
LIN {X 99.8253,Y -89.6591,Z 172,A -39.7831,B 9.2723,C 0.3001,E1 9.3971,E2 490.984} C_DIS
LIN {X 102.4578,Y -86.6381,Z 172,A -37.9117,B 9.2725,C 0.2926,E1 9.4006,E2 489.0907} C_DIS
LIN {X 105.3466,Y -83.1023,Z 172,A -36.1616,B 9.2725,C 0.2926,E1 9.4036,E2 487.3636} C_DIS
LIN {X 108.3224,Y -79.1844,Z 172,A -33.4828,B 9.2731,C 0.2744,E1 9.4082,E2 484.6101} C_DIS
LIN {X 110.9688,Y -75.4308,Z 172,A -31.9706,B 9.2729,C 0.2798,E1 9.4105,E2 483.1523} C_DIS
LIN {X 113.3966,Y -71.7289,Z 172,A -30.2145,B 9.2729,C 0.2781,E1 9.4131,E2 481.4109} C_DIS
LIN {X 115.41,Y -68.443,Z 172,A -28.7684,B 9.2729,C 0.2785,E1 9.4152,E2 479.988} C_DIS
LIN {X 118.0482,Y -63.7848,Z 172,A -26.245,B 9.2733,C 0.2672,E1 9.4186,E2 477.4326} C_DIS
LIN {X 120.3701,Y -59.2816,Z 172,A -23.285,B 9.274,C 0.2431,E1 9.4224,E2 474.3702} C_DIS
LIN {X 123.1729,Y -53.2139,Z 172,A -21.4077,B 9.2736,C 0.2579,E1 9.4244,E2 472.6126} C_DIS
LIN {X 124.5543,Y -49.896,Z 172,A -19.8518,B 9.2736,C 0.2532,E1 9.4261,E2 471.0524} C_DIS
LIN {X 126.1005,Y -45.8486,Z 172,A -18.144,B 9.2737,C 0.2514,E1 9.4277,E2 469.3603} C_DIS
LIN {X 127.0107,Y -43.2649,Z 172,A -16.8391,B 9.2739,C 0.2451,E1 9.4289,E2 468.0375} C_DIS
LIN {X 128.1853,Y -39.6487,Z 172,A -15.4863,B 9.2739,C 0.2467,E1 9.43,E2 466.7165} C_DIS
LIN {X 129.8865,Y -33.6614,Z 172,A -12.5885,B 9.2742,C 0.2337,E1 9.4322,E2 463.7864} C_DIS
LIN {X 130.8947,Y -29.4972,Z 172,A -10.893,B 9.2742,C 0.2316,E1 9.4333,E2 462.1056} C_DIS
LIN {X 131.7216,Y -25.5522,Z 172,A -9.166,B 9.2744,C 0.2265,E1 9.4343,E2 460.3762} C_DIS
LIN {X 132.3965,Y -21.786,Z 172,A -7.4951,B 9.2745,C 0.2209,E1 9.435,E2 458.6989} C_DIS
LIN {X 133.0198,Y -17.5818,Z 172,A -5.8263,B 9.2745,C 0.2191,E1 9.4357,E2 457.0465} C_DIS
LIN {X 133.4317,Y -14.1217,Z 172,A -4.3425,B 9.2746,C 0.2148,E1 9.4361,E2 455.5617} C_DIS
LIN {X 133.7952,Y -10.118,Z 172,A -2.647,B 9.2747,C 0.2103,E1 9.4365,E2 453.8671} C_DIS
LIN {X 134.0571,Y -5.6852,Z 172,A -0.7287,B 9.2749,C 0.2043,E1 9.4368,E2 451.9443} C_DIS
LIN {X 134.1663,Y -1.7504,Z 172,A 0.901,B 9.2749,C 0.2006,E1 9.4369,E2 450.3194} C_DIS
LIN {X 134.1566,Y 2.3359,Z 172,A 2.643,B 9.2751,C 0.1956,E1 9.4369,E2 448.576} C_DIS
LIN {X 134.0237,Y 6.4169,Z 172,A 4.3417,B 9.2751,C 0.1916,E1 9.4367,E2 446.8813} C_DIS
LIN {X 133.7681,Y 10.4886,Z 172,A 6.1264,B 9.2753,C 0.1855,E1 9.4363,E2 445.0898} C_DIS
LIN {X 133.4213,Y 14.2186,Z 172,A 7.6819,B 9.2753,C 0.1819,E1 9.4359,E2 443.5382} C_DIS
LIN {X 132.9037,Y 18.4468,Z 172,A 9.4459,B 9.2754,C 0.178,E1 9.4352,E2 441.7794} C_DIS
LIN {X 132.3241,Y 22.2198,Z 172,A 11.0143,B 9.2754,C 0.1747,E1 9.4345,E2 440.2172} C_DIS
LIN {X 131.613,Y 26.1115,Z 172,A 12.7729,B 9.2756,C 0.1683,E1 9.4336,E2 438.4487} C_DIS
LIN {X 130.8586,Y 29.6552,Z 172,A 14.2554,B 9.2756,C 0.1654,E1 9.4327,E2 436.9728} C_DIS
LIN {X 129.8071,Y 33.968,Z 172,A 16.1563,B 9.2757,C 0.16,E1 9.4314,E2 435.0697} C_DIS
LIN {X 128.7119,Y 37.9028,Z 172,A 18.1636,B 9.2759,C 0.1491,E1 9.4298,E2 433.0286} C_DIS
LIN {X 127.5414,Y 41.6751,Z 172,A 19.4851,B 9.2759,C 0.1528,E1 9.4287,E2 431.7508} C_DIS
LIN {X 124.6159,Y 49.743,Z 172,A 23.0796,B 9.2759,C 0.1445,E1 9.4253,E2 428.1625} C_DIS
LIN {X 123.12,Y 53.3362,Z 172,A 24.649,B 9.276,C 0.1422,E1 9.4235,E2 426.6032} C_DIS
LIN {X 121.9113,Y 56.0445,Z 172,A 25.9433,B 9.276,C 0.1382,E1 9.422,E2 425.3048} C_DIS
LIN {X 120.4631,Y 59.0932,Z 172,A 27.3481,B 9.2761,C 0.1353,E1 9.4203,E2 423.9034} C_DIS
LIN {X 118.9074,Y 62.1638,Z 172,A 28.6025,B 9.2761,C 0.1364,E1 9.4188,E2 422.6745} C_DIS
LIN {X 116.9785,Y 65.7256,Z 172,A 30.6039,B 9.2763,C 0.1259,E1 9.416,E2 420.6389} C_DIS
LIN {X 114.9596,Y 69.1966,Z 172,A 32.2845,B 9.2763,C 0.1225,E1 9.4136,E2 418.9614} C_DIS
LIN {X 112.5957,Y 72.9797,Z 172,A 34.0798,B 9.2763,C 0.1203,E1 9.411,E2 417.1786} C_DIS
LIN {X 110.3438,Y 76.3425,Z 172,A 35.7991,B 9.2763,C 0.1164,E1 9.4083,E2 415.4595} C_DIS
LIN {X 107.8203,Y 79.8667,Z 172,A 37.5088,B 9.2764,C 0.1152,E1 9.4055,E2 413.766} C_DIS
LIN {X 104.9917,Y 83.5497,Z 172,A 39.92,B 9.2766,C 0.1012,E1 9.4013,E2 411.3016} C_DIS
LIN {X 102.6711,Y 86.3857,Z 172,A 41.1865,B 9.2766,C 0.1044,E1 9.399,E2 410.0709} C_DIS
LIN {X 99.6839,Y 89.817,Z 172,A 43.1426,B 9.2766,C 0.0999,E1 9.3954,E2 408.1124} C_DIS
LIN {X 96.9724,Y 92.7371,Z 172,A 44.73,B 9.2766,C 0.0989,E1 9.3924,E2 406.5383} C_DIS
LIN {X 94.4251,Y 95.3297,Z 172,A 46.2704,B 9.2766,C 0.096,E1 9.3894,E2 404.9987} C_DIS
LIN {X 91.37,Y 98.2615,Z 172,A 47.9765,B 9.2766,C 0.0946,E1 9.3859,E2 403.3044} C_DIS
LIN {X 89.0111,Y 100.4036,Z 172,A 49.4674,B 9.2766,C 0.0892,E1 9.3828,E2 401.7973} C_DIS
LIN {X 85.6209,Y 103.3096,Z 172,A 51.3157,B 9.2767,C 0.0869,E1 9.3789,E2 399.9557} C_DIS
LIN {X 82.5683,Y 105.766,Z 172,A 52.8663,B 9.2767,C 0.0866,E1 9.3755,E2 398.4196} C_DIS
LIN {X 79.6581,Y 107.9744,Z 172,A 54.4168,B 9.2767,C 0.0841,E1 9.372,E2 396.8699} C_DIS
LIN {X 75.5712,Y 110.8725,Z 172,A 56.8846,B 9.2768,C 0.0736,E1 9.3663,E2 394.3619} C_DIS
LIN {X 72.757,Y 112.7403,Z 172,A 58.1334,B 9.2768,C 0.0755,E1 9.3634,E2 393.1365} C_DIS
LIN {X 69.5488,Y 114.7467,Z 172,A 59.7713,B 9.2768,C 0.0726,E1 9.3595,E2 391.4957} C_DIS
LIN {X 65.3177,Y 117.2073,Z 172,A 61.8219,B 9.2768,C 0.0705,E1 9.3545,E2 389.4497} C_DIS
LIN {X 61.3042,Y 119.3537,Z 172,A 63.5702,B 9.2768,C 0.072,E1 9.3503,E2 387.725} C_DIS
LIN {X 58.4193,Y 120.7926,Z 172,A 65.1124,B 9.2768,C 0.0669,E1 9.3464,E2 386.1628} C_DIS
LIN {X 55.2241,Y 122.2858,Z 172,A 66.5688,B 9.2768,C 0.0661,E1 9.3427,E2 384.7124} C_DIS
LIN {X 52.0687,Y 123.662,Z 172,A 67.8154,B 9.2768,C 0.0691,E1 9.3395,E2 383.4927} C_DIS
LIN {X 48.6671,Y 125.0392,Z 172,A 69.578,B 9.2768,C 0.0634,E1 9.3349,E2 381.7068} C_DIS
LIN {X 45.7387,Y 126.1401,Z 172,A 71.1015,B 9.2769,C 0.0583,E1 9.3309,E2 380.1607} C_DIS
LIN {X 41.654,Y 127.5494,Z 172,A 73.0677,B 9.2769,C 0.0542,E1 9.3256,E2 378.1803} C_DIS
LIN {X 38.107,Y 128.652,Z 172,A 74.4492,B 9.2769,C 0.0571,E1 9.322,E2 376.8237} C_DIS
LIN {X 33.269,Y 129.9868,Z 172,A 76.4243,B 9.2769,C 0.0589,E1 9.3167,E2 374.8694} C_DIS
LIN {X 30.2052,Y 130.7329,Z 172,A 77.7479,B 9.2769,C 0.0585,E1 9.3131,E2 373.5488} C_DIS
LIN {X 27.0468,Y 131.4226,Z 172,A 79.1178,B 9.2769,C 0.058,E1 9.3094,E2 372.1805} C_DIS
LIN {X 23.9239,Y 132.0269,Z 172,A 80.4587,B 9.2769,C 0.0576,E1 9.3057,E2 370.8422} C_DIS
LIN {X 20.6303,Y 132.5812,Z 172,A 81.7762,B 9.2769,C 0.0592,E1 9.3021,E2 369.5381} C_DIS
LIN {X 17.7947,Y 132.9919,Z 172,A 83.1722,B 9.2769,C 0.0553,E1 9.2982,E2 368.1218} C_DIS
LIN {X 13.9596,Y 133.4492,Z 172,A 84.8407,B 9.2769,C 0.0544,E1 9.2935,E2 366.4515} C_DIS
LIN {X 9.7346,Y 133.8232,Z 172,A 86.591,B 9.2769,C 0.0552,E1 9.2887,E2 364.7092} C_DIS
LIN {X 5.5424,Y 134.0627,Z 172,A 88.2359,B 9.2769,C 0.0579,E1 9.2842,E2 363.0829} C_DIS
LIN {X 2.0381,Y 134.1615,Z 172,A 89.8495,B 9.2769,C 0.0556,E1 9.2796,E2 361.4559} C_DIS
LIN {X -2.2708,Y 134.1577,Z 172,A 91.7269,B 9.2769,C 0.055,E1 9.2744,E2 359.5748} C_DIS
LIN {X -6.7167,Y 134.0086,Z 172,A 93.6181,B 9.2769,C 0.0554,E1 9.2691,E2 357.6856} C_DIS
LIN {X -10.5636,Y 133.7623,Z 172,A 95.3812,B 9.2769,C 0.0535,E1 9.2641,E2 355.9093} C_DIS
LIN {X -14.499,Y 133.3911,Z 172,A 96.9063,B 9.2769,C 0.0572,E1 9.26,E2 354.4048} C_DIS
LIN {X -18.1978,Y 132.9391,Z 172,A 98.6448,B 9.2769,C 0.055,E1 9.2551,E2 352.6495} C_DIS
LIN {X -21.7671,Y 132.3996,Z 172,A 100.1342,B 9.2769,C 0.0568,E1 9.251,E2 351.1672} C_DIS
LIN {X -25.6419,Y 131.7044,Z 172,A 101.7444,B 9.2769,C 0.059,E1 9.2466,E2 349.5666} C_DIS
LIN {X -29.3995,Y 130.917,Z 172,A 103.4092,B 9.2769,C 0.0596,E1 9.2421,E2 347.8998} C_DIS
LIN {X -32.4008,Y 130.2072,Z 172,A 104.8251,B 9.2769,C 0.0587,E1 9.2382,E2 346.4729} C_DIS
LIN {X -41.5195,Y 127.593,Z 172,A 108.9038,B 9.2769,C 0.0617,E1 9.2273,E2 342.394} C_DIS
LIN {X -49.4959,Y 124.7152,Z 172,A 112.5219,B 9.2769,C 0.0655,E1 9.2178,E2 338.779} C_DIS
LIN {X -53.0938,Y 123.2249,Z 172,A 113.9907,B 9.2769,C 0.071,E1 9.2141,E2 337.3348} C_DIS
LIN {X -56.0677,Y 121.9006,Z 172,A 115.4691,B 9.2769,C 0.071,E1 9.2103,E2 335.8469} C_DIS
LIN {X -61.9379,Y 119.0261,Z 172,A 118.3645,B 9.2769,C 0.0729,E1 9.2031,E2 332.9415} C_DIS
LIN {X -65.8316,Y 116.9189,Z 172,A 120.2961,B 9.2769,C 0.0749,E1 9.1983,E2 331.0066} C_DIS
LIN {X -69.554,Y 114.7435,Z 172,A 122.4194,B 9.2769,C 0.0726,E1 9.1931,E2 328.851} C_DIS
LIN {X -72.5233,Y 112.8904,Z 172,A 123.628,B 9.2768,C 0.0801,E1 9.1904,E2 327.6781} C_DIS
LIN {X -75.5023,Y 110.9204,Z 172,A 125.2995,B 9.2768,C 0.0801,E1 9.1865,E2 325.9904} C_DIS
LIN {X -82.2881,Y 105.9834,Z 172,A 128.7671,B 9.2767,C 0.0884,E1 9.1787,E2 322.5402} C_DIS
LIN {X -85.3038,Y 103.5722,Z 172,A 130.4965,B 9.2767,C 0.0901,E1 9.175,E2 320.8027} C_DIS
LIN {X -87.4755,Y 101.7441,Z 172,A 131.9626,B 9.2767,C 0.088,E1 9.1718,E2 319.3071} C_DIS
LIN {X -90.0404,Y 99.4815,Z 172,A 133.1813,B 9.2767,C 0.095,E1 9.1693,E2 318.119} C_DIS
LIN {X -93.0736,Y 96.6501,Z 172,A 135.081,B 9.2767,C 0.0964,E1 9.1655,E2 316.2056} C_DIS
LIN {X -96.601,Y 93.1243,Z 172,A 136.8685,B 9.2765,C 0.1068,E1 9.162,E2 314.4614} C_DIS
LIN {X -99.2195,Y 90.3291,Z 172,A 138.8223,B 9.2765,C 0.1049,E1 9.1583,E2 312.471} C_DIS
LIN {X -102.2269,Y 86.9107,Z 172,A 140.8308,B 9.2765,C 0.1081,E1 9.1546,E2 310.4567} C_DIS
LIN {X -105.2636,Y 83.2079,Z 172,A 142.8739,B 9.2765,C 0.1128,E1 9.151,E2 308.416} C_DIS
LIN {X -107.7441,Y 79.9691,Z 172,A 144.5197,B 9.2764,C 0.1185,E1 9.1483,E2 306.7836} C_DIS
LIN {X -110.5305,Y 76.0712,Z 172,A 146.8794,B 9.2764,C 0.1181,E1 9.1444,E2 304.3882} C_DIS
LIN {X -112.3378,Y 73.377,Z 172,A 148.1317,B 9.2763,C 0.1238,E1 9.1426,E2 303.1534} C_DIS
LIN {X -115.7182,Y 67.92,Z 172,A 150.7455,B 9.2762,C 0.1328,E1 9.1388,E2 300.5578} C_DIS
LIN {X -118.4638,Y 63.0086,Z 172,A 153.2124,B 9.2761,C 0.1379,E1 9.1355,E2 298.0858} C_DIS
LIN {X -120.1576,Y 59.7124,Z 172,A 154.8575,B 9.2761,C 0.141,E1 9.1334,E2 296.4348} C_DIS
LIN {X -121.6963,Y 56.5096,Z 172,A 156.4319,B 9.2761,C 0.1441,E1 9.1315,E2 294.855} C_DIS
LIN {X -123.1729,Y 53.2139,Z 172,A 157.8958,B 9.2759,C 0.1495,E1 9.1299,E2 293.4022} C_DIS
LIN {X -124.521,Y 49.9784,Z 172,A 159.3733,B 9.2759,C 0.1539,E1 9.1283,E2 291.9286} C_DIS
LIN {X -126.5772,Y 44.5183,Z 172,A 161.9956,B 9.2758,C 0.1586,E1 9.1258,E2 289.2932} C_DIS
LIN {X -127.6988,Y 41.1882,Z 172,A 163.5391,B 9.2758,C 0.162,E1 9.1244,E2 287.746} C_DIS
LIN {X -129.0394,Y 36.7776,Z 172,A 165.5376,B 9.2756,C 0.1671,E1 9.1228,E2 285.746} C_DIS
LIN {X -130.0563,Y 32.9953,Z 172,A 167.2252,B 9.2756,C 0.1715,E1 9.1216,E2 284.0582} C_DIS
LIN {X -130.9454,Y 29.2749,Z 172,A 168.9817,B 9.2755,C 0.1742,E1 9.1205,E2 282.2886} C_DIS
LIN {X -131.7637,Y 25.3321,Z 172,A 170.7808,B 9.2755,C 0.1778,E1 9.1195,E2 280.4815} C_DIS
LIN {X -132.5549,Y 20.8003,Z 172,A 172.6285,B 9.2753,C 0.1853,E1 9.1187,E2 278.6499} C_DIS
LIN {X -133.0322,Y 17.4875,Z 172,A 173.9665,B 9.2752,C 0.191,E1 9.1182,E2 277.3244} C_DIS
LIN {X -133.4127,Y 14.2987,Z 172,A 175.482,B 9.2752,C 0.1926,E1 9.1177,E2 275.7928} C_DIS
LIN {X -133.7716,Y 10.4416,Z 172,A 177.2,B 9.2751,C 0.1963,E1 9.1173,E2 274.0687} C_DIS
LIN {X -134.011,Y 6.6682,Z 172,A 178.8238,B 9.275,C 0.2008,E1 9.1171,E2 272.4453} C_DIS
LIN {X -134.1577,Y 2.2708,Z 172,A -179.3019,B 9.2748,C 0.2064,E1 9.1169,E2 270.5734} C_DIS
LIN {X -134.1577,Y -2.2708,Z 172,A -177.2857,B 9.2748,C 0.2108,E1 9.1169,E2 268.5497} C_DIS
LIN {X -134.0161,Y -6.5681,Z 172,A -175.5104,B 9.2746,C 0.2171,E1 9.1172,E2 266.7835} C_DIS
LIN {X -133.8024,Y -10.0193,Z 172,A -173.9299,B 9.2746,C 0.2196,E1 9.1175,E2 265.1916} C_DIS
LIN {X -133.4363,Y -14.0788,Z 172,A -172.14,B 9.2744,C 0.2238,E1 9.118,E2 263.3973} C_DIS
LIN {X -132.9651,Y -17.9998,Z 172,A -170.5188,B 9.2743,C 0.2298,E1 9.1185,E2 261.7856} C_DIS
LIN {X -132.3902,Y -21.8235,Z 172,A -168.8101,B 9.2742,C 0.2335,E1 9.1193,E2 260.0713} C_DIS
LIN {X -131.7418,Y -25.4462,Z 172,A -166.9978,B 9.2742,C 0.234,E1 9.1202,E2 258.2309} C_DIS
LIN {X -130.8517,Y -29.6855,Z 172,A -165.0349,B 9.2742,C 0.2373,E1 9.1214,E2 256.2556} C_DIS
LIN {X -130.0774,Y -32.9122,Z 172,A -163.8391,B 9.2739,C 0.245,E1 9.1222,E2 255.0881} C_DIS
LIN {X -129.181,Y -36.2715,Z 172,A -161.9735,B 9.2739,C 0.2427,E1 9.1237,E2 253.1769} C_DIS
LIN {X -128.032,Y -40.1453,Z 172,A -160.6019,B 9.2737,C 0.2534,E1 9.1247,E2 251.8502} C_DIS
LIN {X -126.7951,Y -43.8898,Z 172,A -158.8401,B 9.2736,C 0.2567,E1 9.1263,E2 250.08} C_DIS
LIN {X -125.1707,Y -48.3289,Z 172,A -156.9319,B 9.2734,C 0.264,E1 9.1282,E2 248.1869} C_DIS
LIN {X -123.9124,Y -51.4691,Z 172,A -155.3659,B 9.2734,C 0.2657,E1 9.1299,E2 246.6069} C_DIS
LIN {X -122.107,Y -55.6213,Z 172,A -152.8133,B 9.2734,C 0.2602,E1 9.1329,E2 243.9793} C_DIS
LIN {X -119.9198,Y -60.1921,Z 172,A -151.3018,B 9.273,C 0.277,E1 9.1346,E2 242.5498} C_DIS
LIN {X -117.0613,Y -65.5782,Z 172,A -148.5267,B 9.273,C 0.2806,E1 9.1384,E2 239.7554} C_DIS
LIN {X -114.7958,Y -69.4675,Z 172,A -146.6169,B 9.2728,C 0.2855,E1 9.1411,E2 237.8481} C_DIS
LIN {X -112.6329,Y -72.9224,Z 172,A -144.4401,B 9.2728,C 0.2821,E1 9.1444,E2 235.6184} C_DIS
LIN {X -110.308,Y -76.3939,Z 172,A -142.9818,B 9.2726,C 0.2919,E1 9.1467,E2 234.2013} C_DIS
LIN {X -107.6211,Y -80.1342,Z 172,A -141.2718,B 9.2723,C 0.3009,E1 9.1494,E2 232.5239} C_DIS
LIN {X -105.2169,Y -83.2668,Z 172,A -139.2717,B 9.2723,C 0.2992,E1 9.1529,E2 230.4859} C_DIS
LIN {X -102.4842,Y -86.608,Z 172,A -137.6271,B 9.2721,C 0.3067,E1 9.1558,E2 228.8667} C_DIS
LIN {X -99.6565,Y -89.8475,Z 172,A -135.2239,B 9.2723,C 0.3005,E1 9.1604,E2 226.3939} C_DIS
LIN {X -96.8933,Y -92.8198,Z 172,A -133.8426,B 9.272,C 0.3103,E1 9.163,E2 225.057} C_DIS
LIN {X -94.8077,Y -94.9496,Z 172,A -132.471,B 9.272,C 0.3111,E1 9.1657,E2 223.6735} C_DIS
LIN {X -92.5676,Y -97.1344,Z 172,A -130.9889,B 9.272,C 0.3111,E1 9.1688,E2 222.1738} C_DIS
LIN {X -90.1668,Y -99.3667,Z 172,A -129.7843,B 9.2717,C 0.3171,E1 9.1712,E2 220.9938} C_DIS
LIN {X -86.6685,Y -102.4328,Z 172,A -127.872,B 9.2716,C 0.3221,E1 9.1752,E2 219.0912} C_DIS
LIN {X -81.9309,Y -106.2603,Z 172,A -125.2397,B 9.2714,C 0.326,E1 9.181,E2 216.4558} C_DIS
LIN {X -76.3957,Y -110.3068,Z 172,A -122.223,B 9.2714,C 0.3291,E1 9.1878,E2 213.4286} C_DIS
LIN {X -72.7766,Y -112.7275,Z 172,A -120.2864,B 9.2713,C 0.3305,E1 9.1924,E2 211.4827} C_DIS
LIN {X -69.194,Y -114.9612,Z 172,A -118.5883,B 9.2711,C 0.335,E1 9.1964,E2 209.7977} C_DIS
LIN {X -65.77,Y -116.9535,Z 172,A -116.8438,B 9.2711,C 0.3362,E1 9.2006,E2 208.0467} C_DIS
LIN {X -62.4718,Y -118.7457,Z 172,A -115.1742,B 9.2711,C 0.337,E1 9.2048,E2 206.3688} C_DIS
LIN {X -58.3373,Y -120.8319,Z 172,A -113.2389,B 9.2709,C 0.3402,E1 9.2096,E2 204.4388} C_DIS
LIN {X -55.0798,Y -122.3503,Z 172,A -111.8605,B 9.2708,C 0.3448,E1 9.213,E2 203.0798} C_DIS
LIN {X -51.6171,Y -123.8506,Z 172,A -110.0584,B 9.2708,C 0.3428,E1 9.2177,E2 201.2539} C_DIS
LIN {X -48.6496,Y -125.046,Z 172,A -108.4398,B 9.271,C 0.3393,E1 9.222,E2 199.6036} C_DIS
LIN {X -45.5185,Y -126.2195,Z 172,A -107.5867,B 9.2705,C 0.3516,E1 9.2241,E2 198.822} C_DIS
LIN {X -41.3058,Y -127.6613,Z 172,A -105.1701,B 9.2708,C 0.3432,E1 9.2306,E2 196.3411} C_DIS
LIN {X -36.642,Y -129.0774,Z 172,A -103.2905,B 9.2706,C 0.3486,E1 9.2356,E2 194.4863} C_DIS
LIN {X -33.1548,Y -130.0158,Z 172,A -101.8962,B 9.2705,C 0.3524,E1 9.2393,E2 193.11} C_DIS
LIN {X -30.0209,Y -130.775,Z 172,A -100.3465,B 9.2705,C 0.3498,E1 9.2436,E2 191.5385} C_DIS
LIN {X -26.1609,Y -131.6029,Z 172,A -98.5561,B 9.2706,C 0.3486,E1 9.2485,E2 189.7346} C_DIS
LIN {X -22.5904,Y -132.2623,Z 172,A -97.1215,B 9.2706,C 0.3514,E1 9.2524,E2 188.314} C_DIS
LIN {X -19.0464,Y -132.818,Z 172,A -95.5984,B 9.2705,C 0.3521,E1 9.2566,E2 186.7914} C_DIS
LIN {X -14.7487,Y -133.3642,Z 172,A -93.7092,B 9.2705,C 0.3517,E1 9.2619,E2 184.8967} C_DIS
LIN {X -11.8503,Y -133.6536,Z 172,A -92.4702,B 9.2705,C 0.352,E1 9.2654,E2 183.6579} C_DIS
LIN {X -8.1574,Y -133.9286,Z 172,A -90.9388,B 9.2705,C 0.3531,E1 9.2696,E2 182.132} C_DIS
LIN {X -3.4453,Y -134.1329,Z 172,A -88.6517,B 9.2707,C 0.3475,E1 9.2761,E2 179.8099} C_DIS
LIN {X 0.9679,Y -134.1726,Z 172,A -87.5376,B 9.2701,C 0.3629,E1 9.2789,E2 178.791} C_DIS
Enddeposition()
LIN {X 0.9679,Y -134.1726,Z 172,A -87.5376,B 9.2701,C 0.3629,E1 9.2789,E2 178.791} C_DIS
Startdeposition()
$VEL.CP = VEL_PRINT
LIN {X 0.2924,Y -135.0865,Z 172,A -88.4006,B 9.008,C 0.3859,E1 9.0151,E2 179.8365} C_DIS
LIN {X -4.4094,Y -135.0156,Z 172,A -89.979,B 9.0084,C 0.3779,E1 9.0108,E2 181.3643} C_DIS
LIN {X -9.3082,Y -134.7659,Z 172,A -91.9765,B 9.0084,C 0.3762,E1 9.0053,E2 183.3523} C_DIS
LIN {X -12.8722,Y -134.4712,Z 172,A -93.3065,B 9.0086,C 0.3724,E1 9.0016,E2 184.6596} C_DIS
LIN {X -16.4572,Y -134.0804,Z 172,A -94.9619,B 9.0086,C 0.3745,E1 8.997,E2 186.3313} C_DIS
LIN {X -20.0473,Y -133.5914,Z 172,A -96.5825,B 9.0085,C 0.3757,E1 8.9925,E2 187.9629} C_DIS
LIN {X -23.913,Y -132.9524,Z 172,A -98.1697,B 9.0085,C 0.3736,E1 8.9881,E2 189.5413} C_DIS
LIN {X -27.6051,Y -132.2368,Z 172,A -99.9091,B 9.0085,C 0.3756,E1 8.9833,E2 191.2991} C_DIS
LIN {X -31.4651,Y -131.3702,Z 172,A -101.4238,B 9.0086,C 0.3716,E1 8.9793,E2 192.7938} C_DIS
LIN {X -34.742,Y -130.5417,Z 172,A -102.875,B 9.0086,C 0.3711,E1 8.9753,E2 194.2475} C_DIS
LIN {X -37.7836,Y -129.6941,Z 172,A -104.1419,B 9.0087,C 0.3688,E1 8.972,E2 195.5058} C_DIS
LIN {X -43.9197,Y -127.747,Z 172,A -107.0157,B 9.0087,C 0.3694,E1 8.9643,E2 198.3978} C_DIS
LIN {X -48.2298,Y -126.1847,Z 172,A -109.1218,B 9.0087,C 0.3706,E1 8.9587,E2 200.5243} C_DIS
LIN {X -52.2261,Y -124.5815,Z 172,A -110.7751,B 9.0089,C 0.3656,E1 8.9545,E2 202.1562} C_DIS
LIN {X -55.9349,Y -122.9637,Z 172,A -112.6617,B 9.0089,C 0.3669,E1 8.9496,E2 204.0641} C_DIS
LIN {X -59.5953,Y -121.2291,Z 172,A -114.4214,B 9.0089,C 0.3657,E1 8.9452,E2 205.8289} C_DIS
LIN {X -64.4352,Y -118.73,Z 172,A -116.6456,B 9.0091,C 0.3612,E1 8.9397,E2 208.0425} C_DIS
LIN {X -68.2609,Y -116.5723,Z 172,A -118.4745,B 9.0091,C 0.3581,E1 8.9353,E2 209.867} C_DIS
LIN {X -70.7938,Y -115.0516,Z 172,A -119.6721,B 9.0093,C 0.3554,E1 8.9325,E2 211.0576} C_DIS
LIN {X -74.0097,Y -113.0101,Z 172,A -121.4561,B 9.0093,C 0.356,E1 8.9282,E2 212.8623} C_DIS
LIN {X -76.9277,Y -111.0442,Z 172,A -123.6171,B 9.0089,C 0.3653,E1 8.9231,E2 215.1052} C_DIS
LIN {X -81.6521,Y -107.6181,Z 172,A -125.4183,B 9.0095,C 0.3495,E1 8.9192,E2 216.8233} C_DIS
LIN {X -86.6443,Y -103.6409,Z 172,A -128.1857,B 9.0097,C 0.3459,E1 8.9132,E2 219.5975} C_DIS
LIN {X -90.1859,Y -100.5739,Z 172,A -130.0843,B 9.0098,C 0.3407,E1 8.9093,E2 221.4847} C_DIS
LIN {X -93.5841,Y -97.4204,Z 172,A -132.0167,B 9.01,C 0.3364,E1 8.9053,E2 223.4123} C_DIS
LIN {X -96.2551,Y -94.7821,Z 172,A -133.7621,B 9.01,C 0.3358,E1 8.9019,E2 225.1761} C_DIS
LIN {X -100.0663,Y -90.7488,Z 172,A -135.9277,B 9.0103,C 0.3278,E1 8.8978,E2 227.3176} C_DIS
LIN {X -102.7512,Y -87.6976,Z 172,A -137.9157,B 9.0103,C 0.3287,E1 8.8941,E2 229.3375} C_DIS
LIN {X -105.6797,Y -84.1452,Z 172,A -139.8393,B 9.0105,C 0.3239,E1 8.8907,E2 231.2567} C_DIS
LIN {X -108.5341,Y -80.4304,Z 172,A -141.9147,B 9.0105,C 0.3209,E1 8.8872,E2 233.342} C_DIS
LIN {X -111.3887,Y -76.4274,Z 172,A -144.3562,B 9.0105,C 0.322,E1 8.8832,E2 235.826} C_DIS
LIN {X -113.6591,Y -73.0087,Z 172,A -145.7765,B 9.0109,C 0.3125,E1 8.8811,E2 237.2062} C_DIS
LIN {X -116.1065,Y -69.0501,Z 172,A -147.7584,B 9.011,C 0.3079,E1 8.8783,E2 239.188} C_DIS
LIN {X -118.0573,Y -65.6594,Z 172,A -149.85,B 9.011,C 0.3108,E1 8.8753,E2 241.3314} C_DIS
LIN {X -120.077,Y -61.8874,Z 172,A -151.2564,B 9.0113,C 0.2996,E1 8.8736,E2 242.6869} C_DIS
LIN {X -121.3704,Y -59.309,Z 172,A -152.8687,B 9.0112,C 0.3028,E1 8.8716,E2 244.3458} C_DIS
LIN {X -123.0748,Y -55.6868,Z 172,A -154.0715,B 9.0116,C 0.2903,E1 8.8702,E2 245.4871} C_DIS
LIN {X -124.5622,Y -52.2723,Z 172,A -155.718,B 9.0116,C 0.2872,E1 8.8684,E2 247.1408} C_DIS
LIN {X -125.8187,Y -49.1712,Z 172,A -157.183,B 9.0118,C 0.2842,E1 8.8669,E2 248.6104} C_DIS
LIN {X -127.0407,Y -45.9214,Z 172,A -158.7395,B 9.0118,C 0.2816,E1 8.8654,E2 250.176} C_DIS
LIN {X -128.371,Y -42.0645,Z 172,A -160.4098,B 9.012,C 0.2759,E1 8.8639,E2 251.8378} C_DIS
LIN {X -129.9596,Y -36.8629,Z 172,A -162.8282,B 9.0122,C 0.2714,E1 8.8619,E2 254.2681} C_DIS
LIN {X -131.5633,Y -30.6525,Z 172,A -165.6312,B 9.0124,C 0.2651,E1 8.86,E2 257.079} C_DIS
LIN {X -132.3532,Y -27.0333,Z 172,A -167.4633,B 9.0124,C 0.2648,E1 8.859,E2 258.9414} C_DIS
LIN {X -132.972,Y -23.8038,Z 172,A -168.5767,B 9.0126,C 0.2564,E1 8.8584,E2 260.0195} C_DIS
LIN {X -133.6328,Y -19.7714,Z 172,A -170.4398,B 9.0126,C 0.2535,E1 8.8576,E2 261.897} C_DIS
LIN {X -134.1151,Y -16.1666,Z 172,A -171.9317,B 9.0128,C 0.2483,E1 8.8571,E2 263.3814} C_DIS
LIN {X -134.5347,Y -12.2112,Z 172,A -173.7552,B 9.0129,C 0.2456,E1 8.8566,E2 265.22} C_DIS
LIN {X -134.8134,Y -8.5813,Z 172,A -175.2261,B 9.0131,C 0.24,E1 8.8563,E2 266.6806} C_DIS
LIN {X -135.0067,Y -4.6648,Z 172,A -177.0163,B 9.0131,C 0.2372,E1 8.8561,E2 268.4847} C_DIS
LIN {X -135.0894,Y -0.0354,Z 172,A -179.0548,B 9.0133,C 0.2327,E1 8.8561,E2 270.5305} C_DIS
LIN {X -135.021,Y 4.2149,Z 172,A 179.1705,B 9.0133,C 0.227,E1 8.8561,E2 272.3} C_DIS
LIN {X -134.8315,Y 8.287,Z 172,A 177.5134,B 9.0136,C 0.2208,E1 8.8564,E2 273.9467} C_DIS
LIN {X -134.5385,Y 12.1714,Z 172,A 175.748,B 9.0136,C 0.2179,E1 8.8568,E2 275.7243} C_DIS
LIN {X -134.1345,Y 16.0035,Z 172,A 174.1752,B 9.0138,C 0.2121,E1 8.8573,E2 277.2879} C_DIS
LIN {X -133.5845,Y 20.0922,Z 172,A 172.5102,B 9.0139,C 0.2058,E1 8.8579,E2 278.941} C_DIS
LIN {X -132.8696,Y 24.3759,Z 172,A 170.5459,B 9.0139,C 0.2024,E1 8.8589,E2 280.9183} C_DIS
LIN {X -132.1046,Y 28.224,Z 172,A 168.9113,B 9.0141,C 0.1972,E1 8.8598,E2 282.5476} C_DIS
LIN {X -131.3603,Y 31.5063,Z 172,A 167.6394,B 9.0142,C 0.1907,E1 8.8606,E2 283.7992} C_DIS
LIN {X -130.5529,Y 34.6997,Z 172,A 166.0573,B 9.0142,C 0.1897,E1 8.8617,E2 285.4023} C_DIS
LIN {X -129.6943,Y 37.7829,Z 172,A 164.5961,B 9.0142,C 0.1875,E1 8.8628,E2 286.8747} C_DIS
LIN {X -128.7054,Y 41.0249,Z 172,A 163.1336,B 9.0144,C 0.1839,E1 8.864,E2 288.3386} C_DIS
LIN {X -126.6956,Y 46.8662,Z 172,A 160.2752,B 9.0144,C 0.1805,E1 8.8667,E2 291.223} C_DIS
LIN {X -124.7942,Y 51.7169,Z 172,A 158.3333,B 9.0146,C 0.1702,E1 8.8687,E2 293.1304} C_DIS
LIN {X -123.4379,Y 54.875,Z 172,A 156.7727,B 9.0146,C 0.1679,E1 8.8704,E2 294.7019} C_DIS
LIN {X -122.1061,Y 57.7791,Z 172,A 155.3615,B 9.0147,C 0.1653,E1 8.8721,E2 296.1184} C_DIS
LIN {X -120.4931,Y 61.0699,Z 172,A 153.7622,B 9.0147,C 0.1619,E1 8.8741,E2 297.7214} C_DIS
LIN {X -116.9696,Y 67.5777,Z 172,A 150.51,B 9.0149,C 0.1557,E1 8.8785,E2 300.9841} C_DIS
LIN {X -114.7226,Y 71.3256,Z 172,A 148.6183,B 9.0149,C 0.1517,E1 8.8812,E2 302.8785} C_DIS
LIN {X -112.217,Y 75.2065,Z 172,A 146.904,B 9.0151,C 0.1429,E1 8.8838,E2 304.5614} C_DIS
LIN {X -109.3926,Y 79.2583,Z 172,A 144.528,B 9.0151,C 0.1425,E1 8.8877,E2 306.969} C_DIS
LIN {X -106.649,Y 82.9134,Z 172,A 142.6179,B 9.0151,C 0.1375,E1 8.8909,E2 308.8738} C_DIS
LIN {X -104.0443,Y 86.1592,Z 172,A 140.7903,B 9.0152,C 0.1345,E1 8.8941,E2 310.707} C_DIS
LIN {X -101.2639,Y 89.4105,Z 172,A 139.1346,B 9.0153,C 0.1278,E1 8.8971,E2 312.342} C_DIS
LIN {X -99.086,Y 91.8184,Z 172,A 137.4565,B 9.0153,C 0.1298,E1 8.9004,E2 314.0547} C_DIS
LIN {X -95.6959,Y 95.3464,Z 172,A 135.5433,B 9.0154,C 0.1228,E1 8.9041,E2 315.9465} C_DIS
LIN {X -93.3394,Y 97.6543,Z 172,A 134.0382,B 9.0154,C 0.1217,E1 8.9071,E2 317.4629} C_DIS
LIN {X -90.0781,Y 100.6705,Z 172,A 131.9213,B 9.0154,C 0.1218,E1 8.9115,E2 319.6057} C_DIS
LIN {X -87.6611,Y 102.7823,Z 172,A 130.7343,B 9.0154,C 0.1163,E1 8.914,E2 320.7707} C_DIS
LIN {X -84.3038,Y 105.5535,Z 172,A 128.8767,B 9.0155,C 0.1131,E1 8.918,E2 322.6278} C_DIS
LIN {X -79.4922,Y 109.2225,Z 172,A 125.8492,B 9.0155,C 0.1163,E1 8.9249,E2 325.7077} C_DIS
LIN {X -75.8539,Y 111.7802,Z 172,A 124.3637,B 9.0156,C 0.1064,E1 8.9282,E2 327.1439} C_DIS
LIN {X -72.1161,Y 114.2273,Z 172,A 122.5999,B 9.0156,C 0.1012,E1 8.9323,E2 328.8905} C_DIS
LIN {X -69.2653,Y 115.9782,Z 172,A 120.8634,B 9.0156,C 0.1044,E1 8.9366,E2 330.6635} C_DIS
LIN {X -64.6088,Y 118.6353,Z 172,A 118.9852,B 9.0157,C 0.0943,E1 8.941,E2 332.4927} C_DIS
LIN {X -61.0119,Y 120.5226,Z 172,A 116.5678,B 9.0157,C 0.104,E1 8.9472,E2 334.9911} C_DIS
LIN {X -56.9935,Y 122.4742,Z 172,A 115.1548,B 9.0157,C 0.0933,E1 8.9507,E2 336.3455} C_DIS
LIN {X -53.8763,Y 123.877,Z 172,A 113.6723,B 9.0157,C 0.0921,E1 8.9545,E2 337.8307} C_DIS
LIN {X -50.173,Y 125.4228,Z 172,A 111.0543,B 9.0157,C 0.1062,E1 8.9616,E2 340.5557} C_DIS
LIN {X -43.8599,Y 127.7677,Z 172,A 109.0178,B 9.0157,C 0.089,E1 8.9666,E2 342.4934} C_DIS
LIN {X -40.1172,Y 128.9926,Z 172,A 106.6499,B 9.0157,C 0.0999,E1 8.9732,E2 344.9427} C_DIS
LIN {X -34.4237,Y 130.6265,Z 172,A 104.8163,B 9.0158,C 0.0859,E1 8.9779,E2 346.6944} C_DIS
LIN {X -30.2855,Y 131.6472,Z 172,A 103.1397,B 9.0158,C 0.0822,E1 8.9824,E2 348.354} C_DIS
LIN {X -26.9833,Y 132.3633,Z 172,A 101.6904,B 9.0158,C 0.0816,E1 8.9863,E2 349.8044} C_DIS
LIN {X -23.7886,Y 132.9747,Z 172,A 100.3421,B 9.0158,C 0.0803,E1 8.99,E2 351.1481} C_DIS
LIN {X -20.6555,Y 133.4973,Z 172,A 98.9418,B 9.0158,C 0.0806,E1 8.9939,E2 352.554} C_DIS
LIN {X -16.9513,Y 134.0194,Z 172,A 97.3494,B 9.0158,C 0.0801,E1 8.9983,E2 354.1462} C_DIS
LIN {X -13.0807,Y 134.4512,Z 172,A 95.6865,B 9.0158,C 0.0797,E1 9.0029,E2 355.8094} C_DIS
LIN {X -9.0459,Y 134.7848,Z 172,A 93.9392,B 9.0158,C 0.0799,E1 9.0078,E2 357.5595} C_DIS
LIN {X -5.331,Y 134.9808,Z 172,A 92.4109,B 9.0158,C 0.0787,E1 9.0121,E2 359.081} C_DIS
LIN {X -1.6122,Y 135.0779,Z 172,A 90.7897,B 9.0158,C 0.0794,E1 9.0166,E2 360.7068} C_DIS
LIN {X 2.0882,Y 135.07,Z 172,A 89.242,B 9.0158,C 0.079,E1 9.0209,E2 362.2511} C_DIS
LIN {X 6.0343,Y 134.9532,Z 172,A 87.5873,B 9.0158,C 0.0788,E1 9.0255,E2 363.9028} C_DIS
LIN {X 9.1803,Y 134.7752,Z 172,A 86.1391,B 9.0158,C 0.0811,E1 9.0296,E2 365.3638} C_DIS
LIN {X 12.7522,Y 134.4827,Z 172,A 84.7243,B 9.0158,C 0.0794,E1 9.0335,E2 366.7654} C_DIS
LIN {X 16.6824,Y 134.0535,Z 172,A 82.9455,B 9.0158,C 0.0819,E1 9.0385,E2 368.5559} C_DIS
LIN {X 20.6519,Y 133.4978,Z 172,A 81.3472,B 9.0158,C 0.0806,E1 9.0428,E2 370.1414} C_DIS
LIN {X 24.3171,Y 132.8801,Z 172,A 79.7049,B 9.0158,C 0.0827,E1 9.0474,E2 371.7911} C_DIS
LIN {X 28.3347,Y 132.0807,Z 172,A 78.0034,B 9.0158,C 0.083,E1 9.052,E2 373.4878} C_DIS
LIN {X 32.5818,Y 131.0992,Z 172,A 76.0931,B 9.0158,C 0.0854,E1 9.0572,E2 375.4051} C_DIS
LIN {X 36.0508,Y 130.1867,Z 172,A 74.0488,B 9.0158,C 0.0967,E1 9.0629,E2 377.5114} C_DIS
LIN {X 40.9574,Y 128.727,Z 172,A 72.5649,B 9.0158,C 0.085,E1 9.0666,E2 378.913} C_DIS
LIN {X 44.0172,Y 127.7132,Z 172,A 71.2071,B 9.0158,C 0.0861,E1 9.0702,E2 380.2695} C_DIS
LIN {X 47.6653,Y 126.397,Z 172,A 69.5501,B 9.0158,C 0.0879,E1 9.0746,E2 381.9278} C_DIS
LIN {X 50.7881,Y 125.1749,Z 172,A 68.0195,B 9.0158,C 0.0916,E1 9.0786,E2 383.4713} C_DIS
LIN {X 54.9359,Y 123.4107,Z 172,A 66.2097,B 9.0158,C 0.0917,E1 9.0832,E2 385.2687} C_DIS
LIN {X 57.7949,Y 122.0985,Z 172,A 64.9171,B 9.0158,C 0.0925,E1 9.0864,E2 386.5563} C_DIS
LIN {X 60.9843,Y 120.5367,Z 172,A 63.3672,B 9.0158,C 0.0953,E1 9.0903,E2 388.1114} C_DIS
LIN {X 64.3785,Y 118.7609,Z 172,A 61.6683,B 9.0157,C 0.099,E1 9.0945,E2 389.8194} C_DIS
LIN {X 67.8161,Y 116.8316,Z 172,A 60.1743,B 9.0157,C 0.0977,E1 9.0981,E2 391.2921} C_DIS
LIN {X 70.8936,Y 114.9905,Z 172,A 58.5274,B 9.0157,C 0.1025,E1 9.1021,E2 392.9543} C_DIS
LIN {X 74.2553,Y 112.8484,Z 172,A 56.4258,B 9.0155,C 0.1136,E1 9.1071,E2 395.1054} C_DIS
LIN {X 77.9739,Y 110.3118,Z 172,A 54.9592,B 9.0155,C 0.1076,E1 9.1103,E2 396.5192} C_DIS
LIN {X 81.6683,Y 107.606,Z 172,A 53.2887,B 9.0156,C 0.1053,E1 9.114,E2 398.1573} C_DIS
LIN {X 84.3628,Y 105.5065,Z 172,A 51.5997,B 9.0156,C 0.1129,E1 9.1178,E2 399.8756} C_DIS
LIN {X 87.8248,Y 102.6431,Z 172,A 49.7892,B 9.0156,C 0.1144,E1 9.1216,E2 401.6751} C_DIS
LIN {X 90.9755,Y 99.8606,Z 172,A 48.0244,B 9.0155,C 0.1174,E1 9.1253,E2 403.4383} C_DIS
LIN {X 93.8733,Y 97.1413,Z 172,A 46.284,B 9.0155,C 0.1219,E1 9.1288,E2 405.1857} C_DIS
LIN {X 97.3078,Y 93.7013,Z 172,A 44.31,B 9.0154,C 0.1242,E1 9.1327,E2 407.1499} C_DIS
LIN {X 100.218,Y 90.5816,Z 172,A 42.4662,B 9.0154,C 0.1288,E1 9.1362,E2 408.9984} C_DIS
LIN {X 103.1945,Y 87.1761,Z 172,A 40.668,B 9.0153,C 0.1304,E1 9.1394,E2 410.7829} C_DIS
LIN {X 107.1756,Y 82.2316,Z 172,A 37.8891,B 9.0152,C 0.1383,E1 9.1443,E2 413.5735} C_DIS
LIN {X 109.8688,Y 78.5969,Z 172,A 35.8316,B 9.0151,C 0.1457,E1 9.1477,E2 415.6488} C_DIS
LIN {X 111.7103,Y 75.9572,Z 172,A 34.7054,B 9.0151,C 0.1438,E1 9.1494,E2 416.7467} C_DIS
LIN {X 113.9564,Y 72.5443,Z 172,A 32.9294,B 9.0151,C 0.149,E1 9.1521,E2 418.5288} C_DIS
LIN {X 116.3604,Y 68.6216,Z 172,A 31.1336,B 9.015,C 0.1504,E1 9.1547,E2 420.3068} C_DIS
LIN {X 118.1901,Y 65.4195,Z 172,A 29.4349,B 9.0149,C 0.1572,E1 9.157,E2 422.0228} C_DIS
LIN {X 120.1716,Y 61.7014,Z 172,A 27.7757,B 9.0149,C 0.159,E1 9.1592,E2 423.6675} C_DIS
LIN {X 121.7558,Y 58.5124,Z 172,A 26.3062,B 9.0148,C 0.162,E1 9.161,E2 425.133} C_DIS
LIN {X 123.2346,Y 55.3294,Z 172,A 24.863,B 9.0148,C 0.1649,E1 9.1626,E2 426.5716} C_DIS
Enddeposition()
END
